(* Logix 5000 project; controller P6 vendor 1 type 14 code 92 rev 20.55; software revision 20.01 *)

TASK MainTask (continuous, watchdog 500 ms) : MainProgram

MODULES
   Local : vendor 1 type 14 code 92 (ICP 0, rev 20.55)
      P6_EN2T_PCN : 1756-EN2T (ICP 1, Ethernet 192.168.1.60, rev 10.1)
         P2 : 1756-EN2T (Ethernet 192.168.1.20, rev 10.1, Output RPI 10 ms)
            P2_CONTROLLER : vendor 1 type 14 code 92 (ICP 0, rev 20.1)
         P1 : 1756-EN2T (Ethernet 192.168.1.10, rev 10.1, Output RPI 10 ms)
            P1_CONTROLLER : vendor 1 type 14 code 92 (ICP 0, rev 20.1)
      P6_EN2TR_RIO : vendor 1 type 12 code 200 (ICP 2, Ethernet 192.168.0.60, rev 10.1)
         RIO6 : 1794-AENTR (Ethernet 192.168.0.62, rev 1.1, Output RPI 20 ms)
            RIO6_DI : 1794-IB32 (Flex 0, rev 1.1, Input RPI 20 ms)
            RIO6_DO : vendor 1 type 7 code 35 (Flex 1, rev 1.1)
            RIO6_AI : 1794-IE12 (Flex 2, rev 1.1, Output RPI 78 ms)
         WRIO6 : vendor 309 type 12 code 1000 (Ethernet 192.168.0.65, rev 3.1, Output RPI 20 ms)
            WRIO6_AI : 1734-IE2C (PointIO 1, rev 3.1, Input RPI 80 ms)
END_MODULES

TYPE AIN_UDT :
STRUCT
   Pv : REAL;
   Heu : REAL;
   Leu : REAL;
   SAHH : REAL;
   SAH : REAL;
   SAL : REAL;
   SALL : REAL;
   AHH : BOOL;
   AH : BOOL;
   AL : BOOL;
   ALL : BOOL;
   Wifi_Enb : BOOL;
   Hty : BOOL;
   Sim : BOOL;
   Sim_PV : REAL;
END_STRUCT
END_TYPE

TYPE AUTOINP_UDT :
STRUCT
   ON : BOOL;
END_STRUCT
END_TYPE

TYPE ControllerLEDStatus :
STRUCT
   Off : BOOL;
   SolidGreen : BOOL;
   FlashingGreen : BOOL;
   SolidYellow : BOOL;
   FlashingYellow : BOOL;
   FlashingRed : BOOL;
   SolidRed : BOOL;
END_STRUCT
END_TYPE

TYPE DOSING_SETPOINT_UDT :
STRUCT
   High_Setpoint : REAL;
   Low_Setpoint : REAL;
END_STRUCT
END_TYPE

TYPE Duty2_UDT :
STRUCT
   Selection : INT;
   Pump_Running : BOOL;
   Selected_Pmp_Not_Avl : BOOL;
   Both_Pmp_Not_Avl : BOOL;
END_STRUCT
END_TYPE

TYPE FaultRecord :
STRUCT
   timelow : DINT;
   timehigh : DINT;
   type : INT;
   code : INT;
   info : DINT[8];
END_STRUCT
END_TYPE

TYPE FIT_UDT :
STRUCT
   Pv : REAL;
   Heu : REAL;
   Leu : REAL;
   SAHH : REAL;
   SAH : REAL;
   SAL : REAL;
   SALL : REAL;
   Totaliser : REAL;
   AHH : BOOL;
   AH : BOOL;
   AL : BOOL;
   ALL : BOOL;
   Sim : BOOL;
   Sim_PV : REAL;
   Wifi_Enb : BOOL;
   Rst_Totaliser : BOOL;
   Hty : BOOL;
END_STRUCT
END_TYPE

TYPE Logix_Status_FP :
STRUCT
   ClearMinorFaults : DINT;
   Sts_MinorFaultEvents : DINT;
   Sts_MinorFaultBits : DINT;
   Sts_Redundant : DINT;
   Set_FaceplateAnimation : DINT;
   Val_ProductCode : DINT;
   MemoryTemp : INT[29];
   Val_raw_data : INT;
   Sts_IO_LED_raw : INT;
   Sts_ProductCode : INT;
   Val_Force_data_raw : INT;
   MemoryRequestData : SINT[12];
   Sts_Force_Installed : BOOL;
   Sts_Force_Enabled : BOOL;
   Sts_Faulted : BOOL;
   Sts_Run : BOOL;
   Sts_Program : BOOL;
   Sts_Minor_fault : BOOL;
   Sts_Major_fault : BOOL;
   Sts_KS_in_run : BOOL;
   Sts_KS_in_program : BOOL;
   Sts_KS_in_remote : BOOL;
   Sts_Changingmodes : BOOL;
   Sts_Test : BOOL;
   Sts_Ladder_Working : BOOL;
   Cmd_ClearFaultRecord : BOOL;
   Set_Controller_Description : STRING;
   UpdateDelayTimer : TIMER;
   Val_MajorFault : FaultRecord;
   Val_MFS : FaultRecord;
   Sts_IO_LED : ControllerLEDStatus;
   Sts_Battery_LED : ControllerLEDStatus;
   MemoryData : Memory_Data;
   TEST : DINT;
END_STRUCT
END_TYPE

TYPE Memory_Data :
STRUCT
   Free_Mem_IO : DINT;
   Free_Mem_DT : DINT;
   Free_Memory : DINT;
   Total_Mem_IO : DINT;
   Total_Mem_DT : DINT;
   Total_Memory : DINT;
   Biggest_IO_Mem_Size_Ava : DINT;
   Biggest_DT_Mem_Size_Ava : DINT;
END_STRUCT
END_TYPE

TYPE MV_UDT :
STRUCT
   Cmd : INT;
   Status : INT;
   Reset : BOOL;
   Auto : BOOL;
   FTO : BOOL;
   FTC : BOOL;
END_STRUCT
END_TYPE

TYPE PLANT_AUTO_UDT :
STRUCT
   ON : BOOL;
   OFF : BOOL;
END_STRUCT
END_TYPE

TYPE PLANT_UDT :
STRUCT
   START : BOOL;
   STOP : BOOL;
END_STRUCT
END_TYPE

TYPE PMP_UDT :
STRUCT
   Cmd : INT;
   Status : INT;
   RunMin : REAL;
   Total_RunMin : REAL;
   RunHr : REAL;
   Total_RunHr : REAL;
   Remote : BOOL;
   Auto : BOOL;
   Fault : BOOL;
   Avl : BOOL;
   Permissive : DINT;
   Shutdown : DINT;
   SD : DINT;
   Reset : BOOL;
   Reset_RunHr : BOOL;
   FTR : BOOL;
   FTS : BOOL;
END_STRUCT
END_TYPE

TYPE PRECONDITION_UDT :
STRUCT
   PERMISSIVE1 : BOOL;
   PERMISSIVE2 : BOOL;
   PERMISSIVE3 : BOOL;
   PERMISSIVE4 : BOOL;
   PERMISSIVE5 : BOOL;
   SHUTDOWN1 : BOOL;
   SHUTDOWN2 : BOOL;
   SHUTDOWN3 : BOOL;
   SHUTDOWN4 : BOOL;
   SHUTDOWN5 : BOOL;
END_STRUCT
END_TYPE

TYPE RED_STAT :
STRUCT
   Redundancy_status_of_the_controller : INT;
   Redundancy_state_of_the_partner : INT;
END_STRUCT
END_TYPE

TYPE SWITCH_UDT :
STRUCT
   Alarm : BOOL;
   Delay : DINT;
END_STRUCT
END_TYPE

TYPE UV_UDT :
STRUCT
   Cmd : INT;
   Status : INT;
   RunMin : REAL;
   Total_RunMin : REAL;
   RunHr : REAL;
   Total_RunHr : REAL;
   Remote : BOOL;
   Auto : BOOL;
   Fault : BOOL;
   Avl : BOOL;
   Permissive : INT;
   Shutdown : INT;
   Reset : BOOL;
   Reset_RunHr : BOOL;
   FT_Start : BOOL;
   FT_Stop : BOOL;
END_STRUCT
END_TYPE

TYPE WIFI_UDT :
STRUCT
   PLC_WIFI : BOOL;
   RIO_WIFI : BOOL;
END_STRUCT
END_TYPE

ADD_ON_INSTRUCTION AIN_FBD   (* revision 1.0 *)
VAR_INPUT
   WRIO_Enb : BOOL; {visible}
   Raw_RIO : INT; {visible}
   Raw_WRIO : INT; {visible}
   L_Raw_RIO : INT; {visible}
   H_Raw_RIO : INT; {visible}
   L_Raw_WRIO : INT; {visible}
   H_Raw_WRIO : INT; {visible}
   HEU : INT; {visible}
   LEU : INT; {visible}
END_VAR
VAR_OUTPUT
   Hty : BOOL; {visible}
   Wifi_Enb : BOOL; {access Read Only, visible}
   AHH : BOOL; {visible}
   AH : BOOL; {access Read Only, visible}
   AL : BOOL; {access Read Only, visible}
   ALL : BOOL; {visible}
END_VAR
VAR_INPUT
   SAHH : REAL; {visible}
   SAH : REAL; {visible}
   SAL : REAL; {visible}
   SALL : REAL; {visible}
   Simulation : BOOL; {visible}
   RIO_Hty : BOOL; {visible}
   WRIO_Hty : BOOL; {visible}
END_VAR
VAR_IN_OUT
   Pv : REAL; {required}
   Sim_PV : REAL; {required}
   HMI : AIN_UDT; {required}
END_VAR
VAR
   SCALE : SCALE; {access None}
   ALM : ALARM; {access None}
   _Raw : INT; {access None}
   _L_Raw : INT; {access None}
   _H_Raw : INT; {access None}
   _Inst_Hty : BOOL; {access None}
END_VAR

ROUTINE Logic   (* structured text *)
   (*RIO and Wireless RIO Selection*)
   
   IF WRIO_Enb THEN
   	Wifi_Enb	:= 1;
   	_Raw		:= Raw_WRIO;
   	_H_Raw		:= H_Raw_WRIO;
   	_L_Raw		:= L_Raw_WRIO;
   	_Inst_Hty 	:= WRIO_Hty;
   ELSE
   	Wifi_Enb	:= 0;
   	_Raw		:= Raw_RIO;
   	_H_Raw		:= H_Raw_RIO;
   	_L_Raw		:= L_Raw_RIO;
   	_Inst_Hty 	:= RIO_Hty;
   END_IF;
   
   (*Calculation for PV*)
   IF Simulation THEN
   	Pv	:=Sim_PV;
   ELSE
   	SCALE.In		:=_Raw;
   	SCALE.InRawMax	:=_H_Raw;
   	SCALE.InRawMin	:=_L_Raw;
   	SCALE.InEUMax	:=HEU;
   	SCALE.InEUMin	:=LEU;
   	SCL(SCALE);
   
   	IF SCALE.Out<0 THEN
   		Pv	:= 0.0;
   	ELSE
   		Pv	:=SCALE.Out;
   	END_IF;
   
   	Sim_PV	:=Pv;
   
   END_IF;
   
   (*Alarms*)
   ALM.In			:=Pv;
   ALM.HHLimit		:=SAHH;
   ALM.HLimit		:=SAH;
   ALM.LLimit		:=SAL;
   ALM.LLLimit		:=SALL;
   ALM(ALM);
   
   AHH				:=ALM.HHAlarm;
   AH				:=ALM.HAlarm;
   AL				:=ALM.LAlarm;
   ALL				:=ALM.LLAlarm;
   
   Hty:= _Inst_Hty AND (_Raw > _L_Raw) AND (_Raw < _H_Raw)  ;
   
   
   
   
   
   
END_ROUTINE
END_ADD_ON_INSTRUCTION

ADD_ON_INSTRUCTION Duty2_FBD   (* revision 1.0 *)
VAR_INPUT
   AutoInp : BOOL; {visible}
   Selection : INT; {visible}
END_VAR
VAR_OUTPUT
   Start_Pmp1 : BOOL; {visible}
   Start_Pmp2 : BOOL; {visible}
END_VAR
VAR_IN_OUT
   PMP1 : PMP_UDT; {required}
   PMP2 : PMP_UDT; {required}
   HMI : Duty2_UDT; {required}
END_VAR

ROUTINE Logic   (* structured text *)
   IF PMP1.Status=2 OR PMP2.Status=2 THEN
   	HMI.Pump_Running := 1;
   ELSE
   	HMI.Pump_Running := 0;
   END_IF;
   
   HMI.Both_Pmp_Not_Avl		:= NOT PMP1.Avl AND NOT PMP2.Avl;
   
   IF AutoInp THEN
   	CASE Selection OF
   		(*PUMP 1 *)
   		1:
   			IF PMP1.Avl THEN
   				Start_Pmp1					:=1;
   				Start_Pmp2					:=0;
   				HMI.Selected_Pmp_Not_Avl	:=0;
   			ELSIF NOT PMP1.Avl AND PMP2.Avl THEN
   				Start_Pmp1					:=0;
   				Start_Pmp2					:=1;
   				HMI.Selected_Pmp_Not_Avl	:=1;
   			ELSIF NOT PMP1.Avl AND NOT PMP2.Avl	THEN
   				Start_Pmp1					:=0;
   				Start_Pmp2					:=0;
   			ELSE
   				HMI.Selected_Pmp_Not_Avl	:=0;
   			END_IF;
   
   		(*PUMP 2 *)
   		2:
   			IF PMP2.Avl THEN
   				Start_Pmp1					:=0;
   				Start_Pmp2					:=1;
   				HMI.Selected_Pmp_Not_Avl	:=0;
   			ELSIF NOT PMP2.Avl AND PMP1.Avl THEN
   				Start_Pmp1					:=1;
   				Start_Pmp2					:=0;
   				HMI.Selected_Pmp_Not_Avl	:=1;
   			ELSIF NOT PMP1.Avl AND NOT PMP2.Avl	THEN
   				Start_Pmp1					:=0;
   				Start_Pmp2					:=0;
   			ELSE
   				HMI.Selected_Pmp_Not_Avl	:=0;
   			END_IF;
   	END_CASE;
   ELSE
   	Start_Pmp1					:=0;
   	Start_Pmp2					:=0;
   END_IF;
   
   
END_ROUTINE
END_ADD_ON_INSTRUCTION

ADD_ON_INSTRUCTION FIT_FBD   (* revision 1.0 *)
VAR_INPUT
   WRIO_Enb : BOOL; {visible}
   Raw_RIO : INT; {visible}
   Raw_WRIO : INT; {visible}
   L_Raw_RIO : INT; {visible}
   H_Raw_RIO : INT; {visible}
   L_Raw_WRIO : INT; {visible}
   H_Raw_WRIO : INT; {visible}
   HEU : REAL; {visible}
   LEU : REAL; {visible}
END_VAR
VAR_OUTPUT
   Hty : BOOL; {visible}
   Wifi_Enb : BOOL; {visible}
   AHH : BOOL; {visible}
   AH : BOOL; {access Read Only, visible}
   AL : BOOL; {access Read Only, visible}
   ALL : BOOL; {visible}
END_VAR
VAR_INPUT
   SAHH : REAL; {visible}
   SAH : REAL; {visible}
   SAL : REAL; {visible}
   SALL : REAL; {visible}
   Simulation : BOOL; {visible}
   RIO_Hty : BOOL; {visible}
   WRIO_Hty : BOOL; {visible}
   Totaliser_Enb : BOOL; {visible}
   Rst_Totaliser : BOOL; {visible}
END_VAR
VAR_IN_OUT
   Totaliser : REAL; {required}
   Pv : REAL; {required}
   Sim_Pv : REAL; {required}
   HMI : FIT_UDT; {required}
END_VAR
VAR
   SCALE : SCALE; {access None}
   ALM : ALARM; {access None}
   TON : FBD_TIMER; {access None}
   _SEC_P : BOOL; {access None}
   _Inst_Hty : BOOL; {access None}
   _L_Raw : INT; {access None}
   _H_Raw : INT; {access None}
   _Raw : INT; {access None}
   R_TRIG : FBD_ONESHOT; {access None}
END_VAR

ROUTINE Logic   (* structured text *)
   (*RIO and Wireless RIO Selection*)
   
   IF WRIO_Enb THEN
   	Wifi_Enb	:= 1;
   	_Raw		:= Raw_WRIO;
   	_H_Raw		:= H_Raw_WRIO;
   	_L_Raw		:= L_Raw_WRIO;
   	_Inst_Hty 	:= WRIO_Hty;
   ELSE
   	Wifi_Enb	:= 0;
   	_Raw		:= Raw_RIO;
   	_H_Raw		:= H_Raw_RIO;
   	_L_Raw		:= L_Raw_RIO;
   	_Inst_Hty 	:= RIO_Hty;
   END_IF;
   
   (*Calculation for PV*)
   IF Simulation THEN
   	Pv	:= Sim_Pv   ;
   ELSE
   	SCALE.In		:=_Raw;
   	SCALE.InRawMax	:=_H_Raw;
   	SCALE.InRawMin	:=_L_Raw;
   	SCALE.InEUMax	:=HEU;
   	SCALE.InEUMin	:=LEU;
   	SCL(SCALE);
   	IF SCALE.Out>0 THEN
   		Pv	:=SCALE.Out;
   	ELSIF SCALE.Out<=0 THEN
   		Pv	:=0.0;
   	END_IF;
   
   	Sim_Pv	:=Pv;
   END_IF;
   
   (*Alarms*)
   ALM.In			:=Pv;
   ALM.HHLimit		:=SAHH;
   ALM.HLimit		:=SAH;
   ALM.LLimit		:=SAL;
   ALM.LLLimit		:=SALL;
   ALM(ALM);
   
   AHH				:=ALM.HHAlarm;
   AH				:=ALM.HAlarm;
   AL				:=ALM.LAlarm;
   ALL				:=ALM.LLAlarm;
   
   (*SECOND PULSE*)
   TON.PRE	:=1000;
   TON.TimerEnable	:=1;
   TONR(TON );
   R_TRIG.InputBit :=TON.DN ;
   OSRI( R_TRIG);
   _SEC_P  := R_TRIG.OutputBit;
   TON.Reset := _SEC_P;
   
   IF Totaliser_Enb THEN
   	IF _SEC_P THEN
   		HMI.Totaliser := HMI.Totaliser +  (ABS(Pv) / 3600 );
   	END_IF;
   END_IF;
   
   IF  Rst_Totaliser   THEN
   	HMI.Totaliser	:=0;
   END_IF;
   
   Hty:= _Inst_Hty AND (_Raw > _L_Raw) AND (_Raw < _H_Raw)  ;
   
   
   
   
   
   
END_ROUTINE
END_ADD_ON_INSTRUCTION

ADD_ON_INSTRUCTION MV_FBD   (* revision 1.0 *)
VAR_INPUT
   Auto : BOOL; {visible}
END_VAR
VAR_OUTPUT
   Cmd_Open : BOOL; {visible}
   Cmd_Close : BOOL; {visible}
   FTO : BOOL; {visible}
   FTC : BOOL; {access Read Only, visible}
END_VAR
VAR_INPUT
   AutoInp : BOOL; {visible}
   ZSO : BOOL; {visible}
   Open_TM : DINT; {visible}
   ZSC : BOOL; {visible}
   Close_TM : DINT; {visible}
END_VAR
VAR_IN_OUT
   Cmd : INT; {required}
   HMI : MV_UDT; {required}
END_VAR
VAR
   TON_Open_TM : FBD_TIMER; {access None}
   TON_Close_TM : FBD_TIMER; {access None}
END_VAR

ROUTINE Logic   (* structured text *)
   (*Fail to Close*)
   TON_Close_TM.PRE 			:= 	Close_TM*1000;
   TON_Close_TM.TimerEnable 	:=  Cmd_Close;
   TONR(TON_Close_TM);
   
   (*Fail to Open*)
   TON_Open_TM.PRE 			:= 	Open_TM*1000;
   TON_Open_TM.TimerEnable 	:= 	Cmd_Open;
   TONR(TON_Open_TM);
   
   IF ZSC THEN
   	HMI.Status	:=1;
   ELSIF ZSO THEN
   	HMI.Status	:=2;
   ELSE
   	HMI.Status	:=0;
   END_IF;
   
   
   IF HMI.Reset THEN
   	(*IF NOT TON_Close_TM.DN AND ZSC THEN*)
   			FTC		:= 0;
   	(*END_IF;*)
   	(*IF NOT TON_Open_TM.DN AND ZSO THEN*)
   			FTO		:= 0;
   	(*END_IF;*)
   END_IF;
   
   IF  NOT Auto THEN
   	CASE HMI.Cmd OF
   		1:	(*CLOSE*)
   			Cmd_Close	:= 1;
   			Cmd_Open	:= 0;
   			IF TON_Close_TM.DN AND (NOT ZSC) THEN
   				FTC		:= 1;
   				FTO		:= 0;
   			END_IF;
   		2:	(*OPEN*)
   			IF FTO OR FTC    THEN
   				HMI.Cmd := 1;
   			END_IF;
   
   			IF NOT FTC AND NOT FTO THEN
   				Cmd_Close	:= 0;
   				Cmd_Open	:= 1;
   			END_IF;
   
   			IF TON_Open_TM.DN AND (NOT ZSO) THEN
   				FTC		:= 0;
   				FTO		:= 1;
   				HMI.Cmd := 1;
   			END_IF;
   	END_CASE;
   ELSE
   	(*Maintain Last status when switching from Auto to Manual*)
   	IF ZSO THEN
   		Cmd	:= 2;
   	END_IF;
   	IF ZSC THEN
   		Cmd	:= 1;
   	END_IF;
   
   	IF  AutoInp  THEN
   		Cmd_Close	:= 0;
   		Cmd_Open	:= 1;
   		IF TON_Open_TM.DN AND (NOT ZSO) THEN
   			FTC		:= 0;
   			FTO		:= 1;
   		END_IF;
   	ELSE
   		Cmd_Close	:= 1;
   		Cmd_Open	:= 0;
   		IF TON_Close_TM.DN AND (NOT ZSC) THEN
   			FTC		:= 1;
   			FTO		:= 0;
   		END_IF;
   	END_IF;
   END_IF;
   
   
END_ROUTINE
END_ADD_ON_INSTRUCTION

ADD_ON_INSTRUCTION PMP_FBD   (* revision 1.0 *)
VAR_OUTPUT
   Cmd_Start : BOOL; {visible}
   Avl : BOOL; {visible}
   Fault : BOOL; {visible}
   FT_Stop : BOOL; {visible}
   FT_Start : BOOL; {visible}
   RunHr : REAL; {visible}
   Total_RunHr : REAL; {visible}
   SD : DINT; {access Read Only, visible}
END_VAR
VAR_INPUT
   Auto : BOOL; {visible}
   AutoInp : BOOL; {visible}
   Remote : BOOL; {visible}
   Run : BOOL; {visible}
   Trip : BOOL; {visible}
   Start_TM : DINT; {visible}
   Stop_TM : DINT; {visible}
   Rst : BOOL; {visible}
   Rst_RunHr : BOOL; {visible}
   Permissive : DINT; {visible}
   Shutdown : DINT; {visible}
END_VAR
VAR_IN_OUT
   RunMin : REAL; {required}
   Total_RunMin : REAL; {required}
   Cmd : INT; {required}
   HMI : PMP_UDT; {required}
END_VAR
VAR
   TON_Start_TM : FBD_TIMER; {access None}
   TON_Stop_TM : FBD_TIMER; {access None}
   _Min_P : BOOL; {access None}
   TON_Min : FBD_TIMER; {access None}
   R_TRIG_SEC : FBD_ONESHOT; {access None}
END_VAR

ROUTINE Logic   (* structured text *)
   (*Fail to Start*)
   TON_Start_TM.PRE 			:= 	Start_TM*1000;
   TON_Start_TM.TimerEnable 	:=  Cmd_Start;
   TONR(TON_Start_TM);
   
   (*Fail to Stop*)
   TON_Stop_TM.PRE 			:= 	Stop_TM*1000;
   TON_Stop_TM.TimerEnable 	:=  NOT Cmd_Start;
   TONR(TON_Stop_TM);
   
   IF (NOT Run) THEN
   	HMI.Status	:=1;
   ELSE
   	HMI.Status	:=2;
   END_IF;
   
   IF Fault THEN
   	HMI.Fault:= 1;
   ELSE
   	HMI.Fault:= 0;
   END_IF;
   
   IF HMI.Reset THEN
   	IF NOT TON_Stop_TM.DN THEN
   			FT_Stop		:= 0;
   	END_IF;
   	IF NOT TON_Start_TM.DN THEN
   			FT_Start	:= 0;
   	END_IF;
   
   	SD :=0;
   
   END_IF;
   
   Fault		:=Trip OR SD<>0;
   HMI.Remote	:=Remote;
   Avl:= Auto AND Remote AND NOT Fault AND NOT FT_Start AND NOT FT_Stop AND SD=0 ;
   
   IF Remote THEN
   	IF  NOT Auto THEN
   		CASE HMI.Cmd OF
   			1:	(*Stop*)
   				Cmd_Start	:=0;
   				IF TON_Stop_TM.DN AND Run THEN
   					FT_Start	:= 0;
   					FT_Stop		:= 1;
   				END_IF;
   			2:	(*OPEN*)
   				IF NOT Fault AND NOT FT_Start AND NOT FT_Stop AND (Permissive=-1) AND HMI.SD=0 THEN
   					Cmd_Start	:= 1;
   				ELSIF Cmd_Start AND (HMI.SD<>0) OR Fault THEN
   					SD				:= HMI.SD;
   					Cmd_Start		:= 0;
   					HMI.Cmd 		:= 1;
   				ELSIF (Permissive<>-1) THEN
   					HMI.Cmd 		:= 1;
   				END_IF;
   
   				IF TON_Start_TM.DN AND NOT Run THEN
   					FT_Start	:= 1;
   					FT_Stop		:= 0;
   					Cmd_Start	:= 0;
   					HMI.Cmd 	:= 1;
   				END_IF;
   		END_CASE;
   	ELSE
   		IF Run THEN
   			Cmd	:= 2;
   		END_IF;
   		IF (NOT Run) OR Fault OR FT_Start OR FT_Stop THEN
   			Cmd	:= 1;
   		END_IF;
   
   		IF  AutoInp  THEN
   			IF NOT Fault AND NOT FT_Start AND NOT FT_Stop AND (Permissive=-1) AND HMI.SD=0  THEN
   				Cmd_Start	:=1;
   			ELSIF Cmd_Start OR (HMI.SD<>0) OR Fault THEN
   				SD			:= HMI.SD;
   				Cmd_Start	:=0;
   			END_IF;
   
   			IF TON_Start_TM.DN AND NOT Run THEN
   				FT_Start	:= 1;
   				FT_Stop		:= 0;
   				Cmd_Start	:= 0;
   				HMI.Cmd 	:= 1;
   			END_IF;
   		ELSE
   			Cmd_Start	:=0;
   			IF TON_Stop_TM.DN AND Run THEN
   				FT_Start	:= 0;
   				FT_Stop		:= 1;
   
   			END_IF;
   		END_IF;
   	END_IF;
   
   ELSE (*Local*)
   	Cmd_Start	:=0;
   	Cmd	:= 1;
   
   	FT_Start	:= 0;
   	FT_Stop		:= 0;
   
   
   
   
   	(*	IF Run THEN
   			Cmd	:= 2;
   		END_IF;
   		IF (NOT Run) OR Fault OR FT_Start OR FT_Stop THEN
   			Cmd	:= 1;
   		END_IF;
   		*)
   END_IF;
   
   (*1 MIN PULSE*)
   TON_Min.PRE	:=60000;
   TON_Min.TimerEnable	:=1;
   TONR(TON_Min );
   R_TRIG_SEC.InputBit :=TON_Min.DN ;
   OSRI( R_TRIG_SEC);
   _Min_P  := R_TRIG_SEC.OutputBit;
   TON_Min.Reset 	:= _Min_P;
   
   IF Run THEN
   	IF _Min_P THEN
   		RunMin 			:=RunMin + 1.0;
   		Total_RunMin	:=Total_RunMin + 1.0;
   	END_IF;
   END_IF;
   
   RunHr 				:=RunMin/60.0;
   Total_RunHr			:=Total_RunMin/60.0;
   
   IF  Rst_RunHr THEN
   	RunMin	:=0;
   END_IF;
   
   
   
END_ROUTINE
END_ADD_ON_INSTRUCTION

ADD_ON_INSTRUCTION SWITCH_FBD   (* revision 1.0 *)
VAR_INPUT
   Alarm : BOOL; {visible}
   Delay : DINT; {required}
END_VAR
VAR_OUTPUT
   Status : BOOL; {access None, required}
END_VAR
VAR_IN_OUT
   HMI : SWITCH_UDT; {required}
END_VAR
VAR
   TON_Delay_Sec : FBD_TIMER; {access None}
END_VAR

ROUTINE Logic   (* structured text *)
   (*Delay for Alarm*)
   TON_Delay_Sec.PRE 			:= 	Delay*1000;
   TON_Delay_Sec.TimerEnable 	:=  Alarm;
   TONR(TON_Delay_Sec);
   
   Status := TON_Delay_Sec.DN ;
END_ROUTINE
END_ADD_ON_INSTRUCTION

ADD_ON_INSTRUCTION UV_FBD   (* revision 1.0 *)
VAR_OUTPUT
   Cmd_Start : BOOL; {visible}
   Avl : BOOL; {visible}
   Fault : BOOL; {visible}
   FT_Stop : BOOL; {visible}
   FT_Start : BOOL; {visible}
   RunHr : REAL; {visible}
   Total_RunHr : REAL; {visible}
END_VAR
VAR_INPUT
   Auto : BOOL; {visible}
   AutoInp : BOOL; {visible}
   Remote : BOOL; {visible}
   Run : BOOL; {visible}
   Trip : BOOL; {visible}
   Start_TM : DINT; {visible}
   Stop_TM : DINT; {visible}
   Rst : BOOL; {visible}
   Rst_RunHr : BOOL; {visible}
   Permissive : INT; {visible}
   Shutdown : INT; {visible}
END_VAR
VAR_IN_OUT
   RunMin : REAL; {required}
   Total_RunMin : REAL; {required}
   Cmd : INT; {required}
   HMI : UV_UDT; {required}
END_VAR
VAR
   TON_Start_TM : FBD_TIMER; {access None}
   TON_Stop_TM : FBD_TIMER; {access None}
   _Min_P : BOOL; {access None}
   TON_Min : FBD_TIMER; {access None}
   R_TRIG_SEC : FBD_ONESHOT; {access None}
END_VAR

ROUTINE Logic   (* structured text *)
   (*Fail to Start*)
   TON_Start_TM.PRE 			:= 	Start_TM*1000;
   TON_Start_TM.TimerEnable 	:=  Cmd_Start;
   TONR(TON_Start_TM);
   
   (*Fail to Stop*)
   TON_Stop_TM.PRE 			:= 	Stop_TM*1000;
   TON_Stop_TM.TimerEnable 	:=  NOT Cmd_Start;
   TONR(TON_Stop_TM);
   
   IF (NOT Run) THEN
   	HMI.Status	:=1;
   ELSE
   	HMI.Status	:=2;
   END_IF;
   
   IF Fault THEN
   	HMI.Fault:= 1;
   ELSE
   	HMI.Fault:= 0;
   END_IF;
   
   IF HMI.Reset THEN
   	IF NOT TON_Stop_TM.DN THEN
   			FT_Stop		:= 0;
   	END_IF;
   	IF NOT TON_Start_TM.DN THEN
   			FT_Start	:= 0;
   	END_IF;
   END_IF;
   
   
   HMI.Remote	:=Remote;
   Avl:= Auto AND Remote AND NOT Fault AND NOT FT_Stop AND NOT FT_Stop   ;
   
   
   
   IF Remote THEN
   	IF  NOT Auto THEN
   		CASE HMI.Cmd OF
   			1:	(*Stop*)
   				Cmd_Start	:=0;
   				IF TON_Stop_TM.DN AND Run THEN
   					FT_Start	:= 0;
   					FT_Stop		:= 1;
   				END_IF;
   			2:	(*OPEN*)
   				IF NOT Fault AND (NOT FT_Start OR FT_Stop) AND (Permissive=-1) THEN
   					Cmd_Start	:= 1;
   				END_IF;
   
   				IF (Shutdown<>0) OR Fault THEN
   					Cmd_Start	:= 0;
   					HMI.Cmd 	:= 1;
   				END_IF;
   
   				IF TON_Start_TM.DN AND NOT Run THEN
   					FT_Start	:= 1;
   					FT_Stop		:= 0;
   					Cmd_Start	:= 0;
   					HMI.Cmd 	:= 1;
   				END_IF;
   		END_CASE;
   	ELSE
   		IF Run THEN
   			Cmd	:= 2;
   		END_IF;
   		IF (NOT Run) OR Fault OR FT_Start OR FT_Stop THEN
   			Cmd	:= 1;
   		END_IF;
   
   		IF  AutoInp  THEN
   			IF NOT Fault AND (NOT FT_Start OR FT_Stop) AND (Permissive=-1) THEN
   				Cmd_Start	:=1;
   			END_IF;
   
   			IF (Shutdown<>0) OR Fault THEN
   				Cmd_Start	:=0;
   			END_IF;
   
   			IF TON_Start_TM.DN AND NOT Run THEN
   				FT_Start	:= 1;
   				FT_Stop		:= 0;
   				Cmd_Start	:= 0;
   				HMI.Cmd 	:= 1;
   			END_IF;
   		ELSE
   			Cmd_Start	:=0;
   			IF TON_Stop_TM.DN AND Run THEN
   				FT_Start	:= 0;
   				FT_Stop		:= 1;
   
   			END_IF;
   		END_IF;
   	END_IF;
   
   ELSE (*Local*)
   	Cmd_Start	:=0;
   	Cmd	:= 1;
   
   	(*	IF Run THEN
   			Cmd	:= 2;
   		END_IF;
   		IF (NOT Run) OR Fault OR FT_Start OR FT_Stop THEN
   			Cmd	:= 1;
   		END_IF;
   		*)
   END_IF;
   
   (*1 MIN PULSE*)
   TON_Min.PRE	:=60000;
   TON_Min.TimerEnable	:=1;
   TONR(TON_Min );
   R_TRIG_SEC.InputBit :=TON_Min.DN ;
   OSRI( R_TRIG_SEC);
   _Min_P  := R_TRIG_SEC.OutputBit;
   TON_Min.Reset 	:= _Min_P;
   
   IF Run THEN
   	IF _Min_P THEN
   		RunMin 			:=RunMin + 1.0;
   		Total_RunMin	:=Total_RunMin + 1.0;
   	END_IF;
   END_IF;
   
   RunHr 				:=RunMin/60.0;
   Total_RunHr			:=Total_RunMin/60.0;
   
   IF  Rst_RunHr THEN
   	RunMin	:=0;
   END_IF;
   
   
   
END_ROUTINE
END_ADD_ON_INSTRUCTION

VAR_GLOBAL   (* controller tags *)
   _FIT601_Tot_Enb : BOOL;
   _MV301_AutoInp : BOOL;
   _MV302_AutoInp : BOOL;
   _MV303_AutoInp : BOOL;
   _MV304_AutoInp : BOOL;
   _P301_AutoInp : BOOL;
   _P302_AutoInp : BOOL;
   _P401_AutoInp : BOOL;
   _P402_AutoInp : BOOL;
   _P403_AutoInp : BOOL;
   _P404_AutoInp : BOOL;
   _P601_AutoInp : BOOL;
   _P602_AutoInp : BOOL;
   _P603_AutoInp : BOOL;
   _P_BACKWASH_SR : DOMINANT_SET;
   _P_CIP_SR : DOMINANT_SET;
   _P_NAHSO3_ORP_DUTY_AutoInp : BOOL;
   _P_NAHSO3_ORP_DUTY_SR : DOMINANT_SET := (Reset := 1, OutNot := 1);
   _P_PERMEATE_SR : DOMINANT_SET := (OutNot := 1);
   _P_RO_FEED_DUTY_AutoInp : BOOL;
   _P_RO_FEED_DUTY_SR : DOMINANT_SET := (Set := 1, Out := 1);
   _P_UF_FEED_DUTY_AutoInp : BOOL := 1;
   _UV401_AutoInp : BOOL := 1;
   _UV_SR : DOMINANT_SET := (Set := 1, Out := 1);
   AI_AIT_401_HRDNSS : INT := -11;
   AI_AIT_401_HRDNSS_HTY : BOOL := 1;
   AI_AIT_402_ORP : INT := -17;
   AI_AIT_402_ORP_HTY : BOOL := 1;
   AI_DPIT_301_DPRESS : INT;
   AI_DPIT_301_DPRESS_HTY : BOOL;
   AI_FIT_301_FLOW : INT;
   AI_FIT_301_FLOW_HTY : BOOL;
   AI_FIT_401_FLOW : INT := -19;
   AI_FIT_401_FLOW_HTY : BOOL := 1;
   AI_FIT_601_FLOW : INT := -3;
   AI_FIT_601_FLOW_HTY : BOOL := 1;
   AI_LIT_301_LEVEL : INT;
   AI_LIT_301_LEVEL_HTY : BOOL;
   AI_LIT_401_LEVEL : INT := -9;
   AI_LIT_401_LEVEL_HTY : BOOL := 1;
   AI_RIO6_SPARE_01 : INT := -7702;
   AI_RIO6_SPARE_01_HTY : BOOL := 1;
   AI_RIO6_SPARE_02 : INT := -7703;
   AI_RIO6_SPARE_02_HTY : BOOL := 1;
   AI_RIO6_SPARE_03 : INT := -7702;
   AI_RIO6_SPARE_03_HTY : BOOL := 1;
   AI_RIO6_SPARE_04 : INT := -7703;
   AI_RIO6_SPARE_04_HTY : BOOL := 1;
   AI_RIO6_SPARE_05 : INT := -7704;
   AI_RIO6_SPARE_05_HTY : BOOL := 1;
   AI_RIO6_SPARE_06 : INT := -7702;
   AI_RIO6_SPARE_06_HTY : BOOL := 1;
   AI_RIO6_SPARE_07 : INT := -7704;
   AI_RIO6_SPARE_07_HTY : BOOL := 1;
   AI_RIO6_SPARE_08 : INT := -7703;
   AI_RIO6_SPARE_08_HTY : BOOL := 1;
   AI_RIO6_SPARE_09 : INT := -7702;
   AI_RIO6_SPARE_09_HTY : BOOL := 1;
   AI_RIO6_SPARE_10 : INT := -7702;
   AI_RIO6_SPARE_10_HTY : BOOL := 1;
   AI_RIO6_SPARE_11 : INT := -7704;
   AI_RIO6_SPARE_11_HTY : BOOL := 1;
   AIT401_FB : AIN_FBD := (Raw_RIO := -11, Raw_WRIO := 3266, H_Raw_RIO := 31208, L_Raw_WRIO := 3277, H_Raw_WRIO := 16383, HEU := 2, Hty := 1, AL := 1, ALL := 1, RIO_Hty := 1);
   AIT401_FB_01 : AIN_FBD;
   AIT402_FB : AIN_FBD := (Raw_RIO := -17, Raw_WRIO := 3268, H_Raw_RIO := 31208, L_Raw_WRIO := 3277, H_Raw_WRIO := 16383, HEU := 2, Hty := 1, AL := 1, ALL := 1, RIO_Hty := 1);
   DI_DPSH_301_HIGH : BOOL;
   DI_LS_401_LOW : BOOL;
   DI_LS_601_HIGH : BOOL := 1;
   DI_LS_601_LOW : BOOL;
   DI_LS_602_HIGH : BOOL := 1;
   DI_LS_602_LOW : BOOL;
   DI_LS_603_HIGH : BOOL;
   DI_LS_603_LOW : BOOL := 1;
   DI_P_404_RUN : BOOL;
   DI_P_601_AUTO : BOOL := 1;
   DI_P_601_FAULT : BOOL;
   DI_P_601_RUN : BOOL;
   DI_P_602_AUTO : BOOL := 1;
   DI_P_602_FAULT : BOOL;
   DI_P_602_RUN : BOOL;
   DI_P_603_AUTO : BOOL := 1;
   DI_P_603_FAULT : BOOL;
   DI_P_603_RUN : BOOL;
   DI_PSH_301_HIGH : BOOL;
   DI_RIO6_SPARE_10 : BOOL;
   DI_RIO6_SPARE_11 : BOOL;
   DI_RIO6_SPARE_12 : BOOL;
   DI_RIO6_SPARE_13 : BOOL;
   DI_RIO6_SPARE_14 : BOOL;
   DI_RIO6_SPARE_15 : BOOL;
   DI_RIO6_SPARE_16 : BOOL;
   DI_RIO6_SPARE_17 : BOOL;
   DI_RIO6_SPARE_18 : BOOL;
   DI_RIO6_SPARE_19 : BOOL;
   DI_RIO6_SPARE_20 : BOOL;
   DI_RIO6_SPARE_21 : BOOL;
   DI_RIO6_SPARE_22 : BOOL;
   DI_RIO6_SPARE_23 : BOOL;
   DI_RIO6_SPARE_24 : BOOL;
   DI_RIO6_SPARE_25 : BOOL;
   DI_RIO6_SPARE_26 : BOOL;
   DI_RIO6_SPARE_27 : BOOL;
   DI_RIO6_SPARE_28 : BOOL;
   DI_RIO6_SPARE_29 : BOOL;
   DI_RIO6_SPARE_30 : BOOL;
   DI_RIO6_SPARE_31 : BOOL;
   DI_UV_401_AUTO : BOOL := 1;
   DI_UV_401_FAULT : BOOL;
   DI_UV_401_RUN : BOOL;
   DI_WIFI_PLC_6 : BOOL;
   DI_WIFI_RIO_6 : BOOL;
   DO_P_601_START : BOOL;
   DO_P_602_START : BOOL;
   DO_P_603_START : BOOL;
   DO_RIO6_SPARE_04 : BOOL;
   DO_RIO6_SPARE_05 : BOOL;
   DO_RIO6_SPARE_06 : BOOL;
   DO_RIO6_SPARE_07 : BOOL;
   DO_RIO6_SPARE_08 : BOOL;
   DO_RIO6_SPARE_09 : BOOL;
   DO_RIO6_SPARE_10 : BOOL;
   DO_RIO6_SPARE_11 : BOOL;
   DO_RIO6_SPARE_12 : BOOL;
   DO_RIO6_SPARE_13 : BOOL;
   DO_RIO6_SPARE_14 : BOOL;
   DO_RIO6_SPARE_15 : BOOL;
   DPIT301_FB : AIN_FBD := (WRIO_Enb := 1, L_Raw_RIO := 6242, H_Raw_RIO := 31208, L_Raw_WRIO := 3277, H_Raw_WRIO := 16383, HEU := 2, Wifi_Enb := 1, AL := 1, ALL := 1);
   DPSH301_FB : SWITCH_FBD;
   FIT102_FB : FIT_FBD;
   FIT301_FB : FIT_FBD := (WRIO_Enb := 1, L_Raw_RIO := 6242, H_Raw_RIO := 31208, L_Raw_WRIO := 3277, H_Raw_WRIO := 16383, HEU := 2.0, Wifi_Enb := 1, AL := 1, ALL := 1);
   FIT401_FB : FIT_FBD := (Raw_RIO := -19, Raw_WRIO := 3263, L_Raw_RIO := 6242, H_Raw_RIO := 31208, L_Raw_WRIO := 3277, H_Raw_WRIO := 16383, HEU := 5.0, Hty := 1, AL := 1, ALL := 1, RIO_Hty := 1);
   FIT601_FB : FIT_FBD := (Raw_RIO := -3, L_Raw_RIO := -5, H_Raw_RIO := 31208, L_Raw_WRIO := 3277, H_Raw_WRIO := 16383, HEU := 2.0, Hty := 1, AL := 1, ALL := 1, SAHH := 3.0, SAH := 2.0, SAL := 1.0, SALL := 0.5, RIO_Hty := 1, WRIO_Hty := 1);
   HMI_AIT202 : AIN_UDT := (Pv := 7.3255577, SAHH := 12.0, SAH := 7.05, SAL := 6.95, SALL := 3.0, AH := 1, Hty := 1, Sim_PV := 7.3255577);
   HMI_FIT301 : FIT_UDT := (Totaliser := -0.09362481, AL := 1, ALL := 1, Wifi_Enb := 1);
   HMI_FIT401 : FIT_UDT := (Pv := -1.2539053, Totaliser := -0.9073935, AL := 1, ALL := 1, Hty := 1);
   HMI_FIT601 : FIT_UDT := (Pv := 0.00012815173, SAHH := 3.0, SAH := 2.0, SAL := 1.0, SALL := 0.5, Totaliser := 0.8749698, AL := 1, ALL := 1, Sim_PV := 0.00012815173, Hty := 1);
   HMI_LIT101 : AIN_UDT := (Pv := 812.6106, SAHH := 1000.0, SAH := 800.0, SAL := 500.0, SALL := 250.0, AH := 1, Hty := 1, Sim_PV := 812.6106);
   HMI_LIT301 : AIN_UDT := (Pv := -0.5000763, AL := 1, ALL := 1, Wifi_Enb := 1);
   HMI_LIT401 : AIN_UDT := (Pv := -0.0005767752, AL := 1, ALL := 1, Hty := 1);
   HMI_LS401 : SWITCH_UDT;
   HMI_LSH601 : SWITCH_UDT := (Alarm := 1);
   HMI_LSH602 : SWITCH_UDT := (Alarm := 1);
   HMI_LSH603 : SWITCH_UDT;
   HMI_LSL601 : SWITCH_UDT;
   HMI_LSL602 : SWITCH_UDT;
   HMI_LSL603 : SWITCH_UDT := (Alarm := 1);
   HMI_NAHSO3_ORP_DOSING : DOSING_SETPOINT_UDT;
   HMI_P301 : PMP_UDT := (Cmd := 1, Status := 1, Remote := 1, Permissive := -1);
   HMI_P302 : PMP_UDT := (Cmd := 1, Status := 1, Remote := 1, Permissive := -1);
   HMI_P401 : PMP_UDT := (Status := 1, Remote := 1, Permissive := -1);
   HMI_P402 : PMP_UDT := (Status := 1, Remote := 1, Permissive := -1);
   HMI_P403 : PMP_UDT := (Status := 1, Remote := 1, Permissive := -1);
   HMI_P404 : PMP_UDT := (Status := 1, Remote := 1, Permissive := -1);
   HMI_P501 : PMP_UDT;
   HMI_P502 : PMP_UDT;
   HMI_P601 : PMP_UDT := (Cmd := 1, Status := 1, RunMin := 2166.0, Total_RunMin := 2166.0, RunHr := 36.1, Total_RunHr := 36.1, Remote := 1, Auto := 1, Avl := 1, Permissive := -1, Reset := 1);
   HMI_P601_MSG : PRECONDITION_UDT := (PERMISSIVE1 := 1);
   HMI_P602 : PMP_UDT := (Cmd := 1, Status := 1, RunMin := 63.0, Total_RunMin := 63.0, RunHr := 1.05, Total_RunHr := 1.05, Remote := 1, Auto := 1, Avl := 1, Permissive := -1, Reset := 1);
   HMI_P602_MSG : PRECONDITION_UDT := (PERMISSIVE1 := 1);
   HMI_P603 : PMP_UDT := (Cmd := 1, Status := 1, Remote := 1, Auto := 1, Avl := 1, Permissive := -2, SD := 1, Reset := 1);
   HMI_P603_MSG : PRECONDITION_UDT;
   HMI_P6_PERMISSIVE : AUTOINP_UDT := (ON := 1);
   HMI_P6_STATE : INT := 1;
   HMI_P_NAHSO3_ORP_DUTY : Duty2_UDT;
   HMI_P_RO_FEED_DUTY : Duty2_UDT;
   HMI_P_UF_FEED_DUTY : Duty2_UDT;
   HMI_PLANT : PLANT_UDT;
   HMI_PLANT_AUTO : PLANT_AUTO_UDT;
   HMI_PLANT_PERMISSIVE : BOOL := 1;
   HMI_PLANT_RESET : PLANT_AUTO_UDT;
   HMI_PSH301 : SWITCH_UDT;
   HMI_START_PLANT : BOOL;
   HMI_STOP_PLANT : BOOL;
   HMI_UV401 : UV_UDT := (Cmd := 1, Status := 1, Remote := 1, Permissive := -1);
   HMI_WIFI : WIFI_UDT;
   LIT301_FB : AIN_FBD := (WRIO_Enb := 1, L_Raw_RIO := 6242, H_Raw_RIO := 31208, L_Raw_WRIO := 3277, H_Raw_WRIO := 16383, HEU := 2, Wifi_Enb := 1, AL := 1, ALL := 1);
   LIT401_FB : AIN_FBD := (Raw_RIO := -9, Raw_WRIO := 3269, H_Raw_RIO := 31208, L_Raw_WRIO := 3277, H_Raw_WRIO := 16383, HEU := 2, Hty := 1, AL := 1, ALL := 1, RIO_Hty := 1);
   LIT401_FB_01 : AIN_FBD;
   Logix_Status : Logix_Status_FP := (Set_FaceplateAnimation := 90, Val_ProductCode := 92, MemoryTemp[0] := 5, MemoryTemp[1] := 1, MemoryTemp[3] := 32290, MemoryTemp[4] := 3, MemoryTemp[5] := 18578, MemoryTemp[6] := 7, MemoryTemp[9] := 2, MemoryTemp[11] := -4608, MemoryTemp[12] := 3, MemoryTemp[14] := 8, MemoryTemp[17] := 5, MemoryTemp[21] := 6, MemoryTemp[23] := 32052, MemoryTemp[24] := 3, MemoryTemp[25] := 7, MemoryTemp[27] := 18376, MemoryTemp[28] := 7, Val_raw_data := 12384, Sts_IO_LED_raw := 2, Sts_ProductCode := 92, MemoryRequestData[0] := 5, MemoryRequestData[2] := 1, MemoryRequestData[4] := 2, MemoryRequestData[6] := 5, MemoryRequestData[8] := 6, MemoryRequestData[10] := 7, Sts_Run := 1, Sts_KS_in_remote := 1, Sts_Ladder_Working := 1, Set_Controller_Description := 'P6: RO Product System', UpdateDelayTimer.PRE := 1000, UpdateDelayTimer.ACC := 798, UpdateDelayTimer.EN := 1, UpdateDelayTimer.TT := 1, Val_MFS.timelow := 71751885, Val_MFS.timehigh := 206334, Val_MFS.type := 3, Val_MFS.code := 20, Val_MFS.info[1] := 1, Sts_IO_LED.FlashingGreen := 1, Sts_Battery_LED.Off := 1, MemoryData.Free_Mem_IO := 915592, MemoryData.Free_Mem_DT := 1909320, MemoryData.Total_Mem_IO := 1030144, MemoryData.Total_Mem_DT := 2097152, MemoryData.Biggest_IO_Mem_Size_Ava := 914640, MemoryData.Biggest_DT_Mem_Size_Ava := 1908512);
   LS401_FB : SWITCH_FBD;
   LSH601_FB : SWITCH_FBD := (Alarm := 1, Status := 1);
   LSH601_FB_01 : SWITCH_FBD;
   LSH601_FB_02 : SWITCH_FBD;
   LSH602_FB : SWITCH_FBD := (Alarm := 1, Status := 1);
   LSH603_FB : SWITCH_FBD;
   LSL601_FB : SWITCH_FBD;
   LSL601_FB_01 : SWITCH_FBD;
   LSL601_FB_02 : SWITCH_FBD;
   LSL601_FB_03 : SWITCH_FBD;
   LSL602_FB : SWITCH_FBD;
   LSL603_FB : SWITCH_FBD := (Alarm := 1, Status := 1);
   Memory_Message : MESSAGE;
        MessageParameters(ServiceCode := 16#0003, LocalElement := Logix_Status.MemoryRequestData[0], DestinationTag := Logix_Status.MemoryTemp[0], ...)
   MV301_FB : MV_FBD := (Cmd_Close := 1, Open_TM := 25, ZSC := 1, Close_TM := 25);
   MV302_FB : MV_FBD := (Cmd_Close := 1, Open_TM := 25, ZSC := 1, Close_TM := 25);
   MV303_FB : MV_FBD := (Cmd_Close := 1, Open_TM := 25, ZSC := 1, Close_TM := 25);
   MV304_FB : MV_FBD := (Cmd_Close := 1, Open_TM := 25, ZSC := 1, Close_TM := 25);
   P1_LIT101_MSG : MESSAGE;
        MessageParameters(ServiceCode := 16#004c, LocalElement := HMI_LIT101, ...)
   P201_FB : PMP_FBD;
   P202_FB : PMP_FBD;
   P2_AIT202_MSG : MESSAGE;
        MessageParameters(ServiceCode := 16#004c, LocalElement := HMI_AIT202, ...)
   P301_FB : PMP_FBD := (Remote := 1, Start_TM := 3, Stop_TM := 3, Permissive := -1);
   P302_FB : PMP_FBD := (Remote := 1, Start_TM := 3, Stop_TM := 3, Permissive := -1);
   P401_FB : PMP_FBD := (Remote := 1, Start_TM := 3, Stop_TM := 3, Permissive := -1);
   P401_FB_01 : PMP_FBD;
   P401_FB_02 : PMP_FBD;
   P402_FB : PMP_FBD := (Remote := 1, Start_TM := 3, Stop_TM := 3, Permissive := -1);
   P402_FB_01 : PMP_FBD;
   P403_FB : PMP_FBD := (Remote := 1, Start_TM := 3, Stop_TM := 3, Permissive := -1);
   P404_FB : PMP_FBD := (Remote := 1, Start_TM := 3, Stop_TM := 3, Permissive := -1);
   P601_FB : PMP_FBD := (Avl := 1, RunHr := 36.1, Total_RunHr := 36.1, Auto := 1, Remote := 1, Start_TM := 3, Stop_TM := 3, Rst := 1, Permissive := -1);
   P601_FB_01 : PMP_FBD;
   P601_FB_02 : PMP_FBD;
   P602_FB : PMP_FBD := (Avl := 1, RunHr := 1.05, Total_RunHr := 1.05, Auto := 1, Remote := 1, Start_TM := 3, Stop_TM := 3, Rst := 1, Permissive := -1);
   P603_FB : PMP_FBD := (Avl := 1, Auto := 1, Remote := 1, Start_TM := 3, Stop_TM := 3, Rst := 1, Permissive := -2, Shutdown := 1);
   P6_P602_AUTOINP : AUTOINP_UDT;
   P_NAHSO3_ORP_DUTY_FB : Duty2_FBD;
   P_RO_FEED_DUTY_FB : Duty2_FBD;
   P_RO_FEED_DUTY_FB_01 : Duty2_FBD;
   P_UF_FEED_DUTY_FB : Duty2_FBD := (AutoInp := 1);
   PLANT_CRITICAL_SD : AUTOINP_UDT;
   PSH301_FB : SWITCH_FBD;
   PSH301_FB_01 : SWITCH_FBD;
   REDUNDANT_STATUS : RED_STAT := (Redundancy_status_of_the_controller := 2, Redundancy_state_of_the_partner := 8);
   UV401_FB : UV_FBD := (AutoInp := 1, Remote := 1, Start_TM := 3, Stop_TM := 3, Permissive := -1);
   W_AI_AIT_401_HRDNSS : INT := 3266;
   W_AI_AIT_401_HRDNSS_HTY : BOOL;
   W_AI_AIT_402_ORP : INT := 3268;
   W_AI_AIT_402_ORP_HTY : BOOL;
   W_AI_DPIT_301_DPRESS : INT;
   W_AI_DPIT_301_DPRESS_HTY : BOOL;
   W_AI_FIT_301_FLOW : INT;
   W_AI_FIT_301_FLOW_HTY : BOOL;
   W_AI_FIT_401_FLOW : INT := 3263;
   W_AI_FIT_401_FLOW_HTY : BOOL;
   W_AI_FIT_601_FLOW : INT;
   W_AI_FIT_601_FLOW_HTY : BOOL := 1;
   W_AI_FIT_601_HTY : BOOL;
   W_AI_LIT_301_LEVEL : INT;
   W_AI_LIT_301_LEVEL_HTY : BOOL;
   W_AI_LIT_401_LEVEL : INT := 3269;
   W_AI_LIT_401_LEVEL_HTY : BOOL;
   W_AI_RIO6_SPARE_01 : INT;
   W_AI_RIO6_SPARE_01_HTY : BOOL := 1;
   XXX : DINT;
END_VAR

PROGRAM MainProgram   (* main routine MainRoutine *)
VAR
   FIT_FBD_01 : FIT_FBD;
   PMP_FBD_01 : PMP_FBD;
   SWITCH_FBD_01 : SWITCH_FBD;
END_VAR

ROUTINE IO   (* structured text *)
   (*DIGITAL INPUTS*)
   DI_WIFI_PLC_6	:=RIO6:0:I.Data.0;
   DI_WIFI_RIO_6	:=RIO6:0:I.Data.1;
   DI_P_601_AUTO	:=RIO6:0:I.Data.2;
   DI_P_601_RUN	:=RIO6:0:I.Data.3;
   DI_P_601_FAULT	:=RIO6:0:I.Data.4;
   DI_P_602_AUTO	:=RIO6:0:I.Data.5;
   DI_P_602_RUN	:=RIO6:0:I.Data.6;
   DI_P_602_FAULT	:=RIO6:0:I.Data.7;
   DI_P_603_AUTO	:=RIO6:0:I.Data.8;
   DI_P_603_RUN	:=RIO6:0:I.Data.9;
   DI_P_603_FAULT	:=RIO6:0:I.Data.10;
   DI_LS_601_LOW	:=RIO6:0:I.Data.11;
   DI_LS_601_HIGH	:=RIO6:0:I.Data.12;
   DI_LS_602_LOW	:=RIO6:0:I.Data.13;
   DI_LS_602_HIGH	:=RIO6:0:I.Data.14;
   DI_LS_603_LOW	:=RIO6:0:I.Data.15;
   DI_LS_603_HIGH	:=RIO6:0:I.Data.16;
   DI_RIO6_SPARE_17:=RIO6:0:I.Data.17;
   DI_RIO6_SPARE_18:=RIO6:0:I.Data.18;
   DI_RIO6_SPARE_19:=RIO6:0:I.Data.19;
   DI_RIO6_SPARE_20:=RIO6:0:I.Data.20;
   DI_RIO6_SPARE_21:=RIO6:0:I.Data.21;
   DI_RIO6_SPARE_22:=RIO6:0:I.Data.22;
   DI_RIO6_SPARE_23:=RIO6:0:I.Data.23;
   DI_RIO6_SPARE_24:=RIO6:0:I.Data.24;
   DI_RIO6_SPARE_25:=RIO6:0:I.Data.25;
   DI_RIO6_SPARE_26:=RIO6:0:I.Data.26;
   DI_RIO6_SPARE_27:=RIO6:0:I.Data.27;
   DI_RIO6_SPARE_28:=RIO6:0:I.Data.28;
   DI_RIO6_SPARE_29:=RIO6:0:I.Data.29;
   DI_RIO6_SPARE_30:=RIO6:0:I.Data.30;
   DI_RIO6_SPARE_31:=RIO6:0:I.Data.31;
   
   (*DIGITAL OUTPUTS*)
   RIO6:1:O.0	:=DO_P_601_START;
   RIO6:1:O.1	:=DO_P_602_START;
   RIO6:1:O.2	:=DO_P_603_START;
   RIO6:1:O.4	:=DO_RIO6_SPARE_04;
   RIO6:1:O.5	:=DO_RIO6_SPARE_05;
   RIO6:1:O.6	:=DO_RIO6_SPARE_06;
   RIO6:1:O.7	:=DO_RIO6_SPARE_07;
   RIO6:1:O.8	:=DO_RIO6_SPARE_08;
   RIO6:1:O.9	:=DO_RIO6_SPARE_09;
   RIO6:1:O.10	:=DO_RIO6_SPARE_10;
   RIO6:1:O.11	:=DO_RIO6_SPARE_11;
   RIO6:1:O.12	:=DO_RIO6_SPARE_12;
   RIO6:1:O.13	:=DO_RIO6_SPARE_13;
   RIO6:1:O.14	:=DO_RIO6_SPARE_14;
   RIO6:1:O.15	:=DO_RIO6_SPARE_15;
   
   (*ANALOG INPUTS*)
   AI_FIT_601_FLOW		:=RIO6:2:I.Ch0Data;
   AI_RIO6_SPARE_01	:=RIO6:2:I.Ch1Data;
   AI_RIO6_SPARE_02	:=RIO6:2:I.Ch2Data;
   AI_RIO6_SPARE_03	:=RIO6:2:I.Ch3Data;
   AI_RIO6_SPARE_04	:=RIO6:2:I.Ch4Data;
   AI_RIO6_SPARE_05	:=RIO6:2:I.Ch5Data;
   AI_RIO6_SPARE_06	:=RIO6:2:I.Ch6Data;
   AI_RIO6_SPARE_07	:=RIO6:2:I.Ch7Data;
   AI_RIO6_SPARE_08	:=RIO6:2:I.Ch8Data;
   AI_RIO6_SPARE_09	:=RIO6:2:I.Ch9Data;
   AI_RIO6_SPARE_10	:=RIO6:2:I.Ch10Data;
   AI_RIO6_SPARE_11	:=RIO6:2:I.Ch11Data;
   
   AI_FIT_601_FLOW_HTY		:=(NOT RIO6:2:I.GeneralFault);
   AI_RIO6_SPARE_01_HTY	:=(NOT RIO6:2:I.GeneralFault);
   AI_RIO6_SPARE_02_HTY	:=(NOT RIO6:2:I.GeneralFault);
   AI_RIO6_SPARE_03_HTY	:=(NOT RIO6:2:I.GeneralFault);
   AI_RIO6_SPARE_04_HTY	:=(NOT RIO6:2:I.GeneralFault);
   AI_RIO6_SPARE_05_HTY	:=(NOT RIO6:2:I.GeneralFault);
   AI_RIO6_SPARE_06_HTY	:=(NOT RIO6:2:I.GeneralFault);
   AI_RIO6_SPARE_07_HTY	:=(NOT RIO6:2:I.GeneralFault);
   AI_RIO6_SPARE_08_HTY	:=(NOT RIO6:2:I.GeneralFault);
   AI_RIO6_SPARE_09_HTY	:=(NOT RIO6:2:I.GeneralFault);
   AI_RIO6_SPARE_10_HTY	:=(NOT RIO6:2:I.GeneralFault);
   AI_RIO6_SPARE_11_HTY	:=(NOT RIO6:2:I.GeneralFault);
   
   (*WIRELESS ANALOG INPUTS*)
   W_AI_FIT_601_FLOW		:=WRIO6:1:I.Ch0Data;
   W_AI_RIO6_SPARE_01		:=WRIO6:1:I.Ch1Data;
   
   W_AI_FIT_601_FLOW_HTY	:=(NOT WRIO6:1:I.Ch0Fault);
   W_AI_RIO6_SPARE_01_HTY	:=(NOT WRIO6:1:I.Ch1Fault);
   
   (*Wireless Selction*)
   HMI_WIFI.PLC_WIFI		:= DI_WIFI_PLC_6;
   HMI_WIFI.RIO_WIFI		:= DI_WIFI_RIO_6;
END_ROUTINE

ROUTINE Logix_Status   (* ladder *)
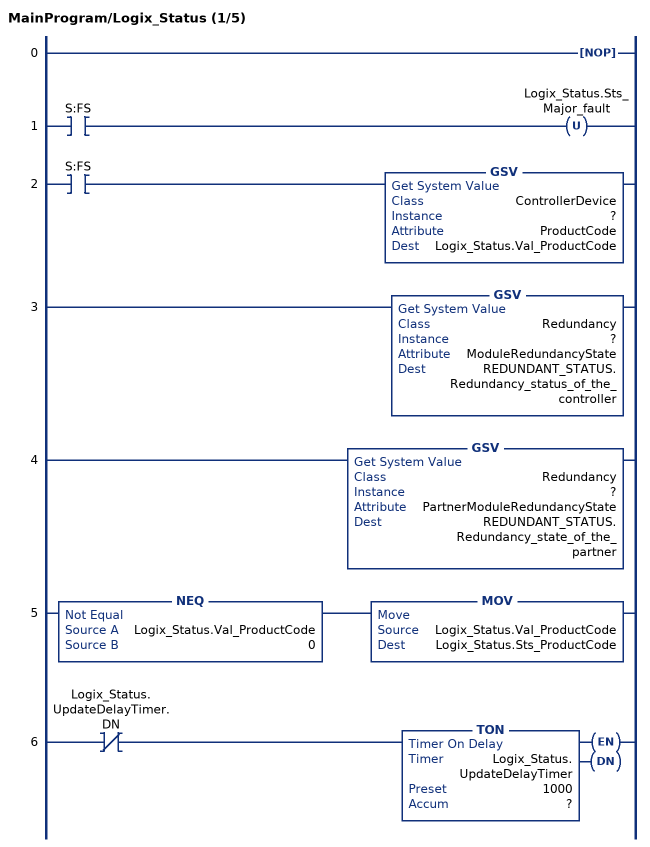
   0: NOP();
   1: XIC(S:FS)OTU(Logix_Status.Sts_Major_fault);
   2: XIC(S:FS)GSV(ControllerDevice,?,ProductCode,Logix_Status.Val_ProductCode);
   3: GSV(Redundancy,?,ModuleRedundancyState,REDUNDANT_STATUS.Redundancy_status_of_the_controller);
   4: GSV(Redundancy,?,PartnerModuleRedundancyState,REDUNDANT_STATUS.Redundancy_state_of_the_partner);
   5: NEQ(Logix_Status.Val_ProductCode,0)MOV(Logix_Status.Val_ProductCode,Logix_Status.Sts_ProductCode);
   6: XIO(Logix_Status.UpdateDelayTimer.DN)TON(Logix_Status.UpdateDelayTimer,?,?);
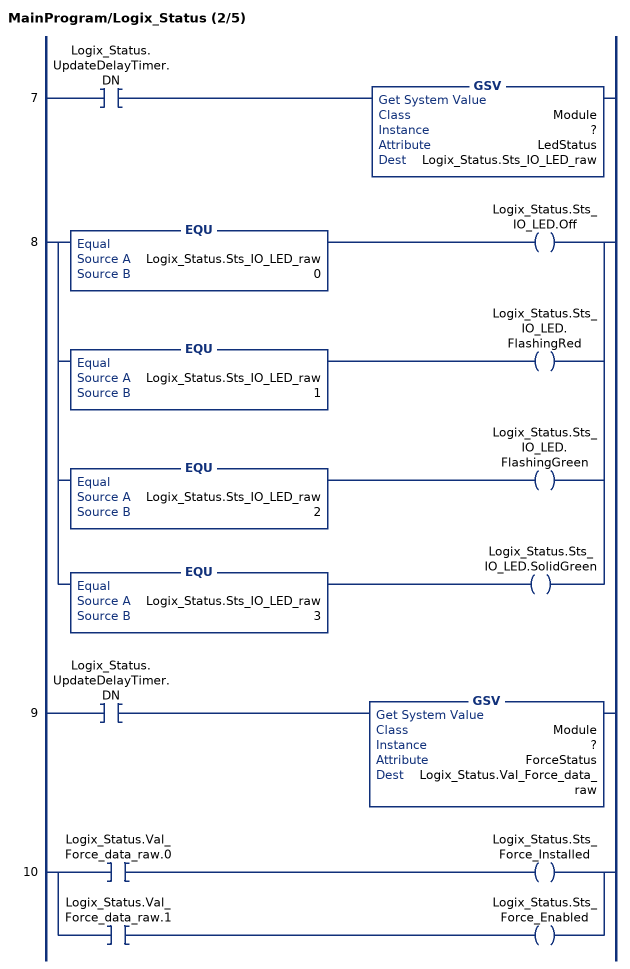
   7: XIC(Logix_Status.UpdateDelayTimer.DN)GSV(Module,?,LedStatus,Logix_Status.Sts_IO_LED_raw);
   8: [EQU(Logix_Status.Sts_IO_LED_raw,0) OTE(Logix_Status.Sts_IO_LED.Off) ,EQU(Logix_Status.Sts_IO_LED_raw,1) OTE(Logix_Status.Sts_IO_LED.FlashingRed) ,EQU(Logix_Status.Sts_IO_LED_raw,2) OTE(Logix_Status.Sts_IO_LED.FlashingGreen) ,EQU(Logix_Status.Sts_IO_LED_raw,3) OTE(Logix_Status.Sts_IO_LED.SolidGreen) ];
   9: XIC(Logix_Status.UpdateDelayTimer.DN)GSV(Module,?,ForceStatus,Logix_Status.Val_Force_data_raw);
   10: [XIC(Logix_Status.Val_Force_data_raw.0) OTE(Logix_Status.Sts_Force_Installed) ,XIC(Logix_Status.Val_Force_data_raw.1) OTE(Logix_Status.Sts_Force_Enabled) ];
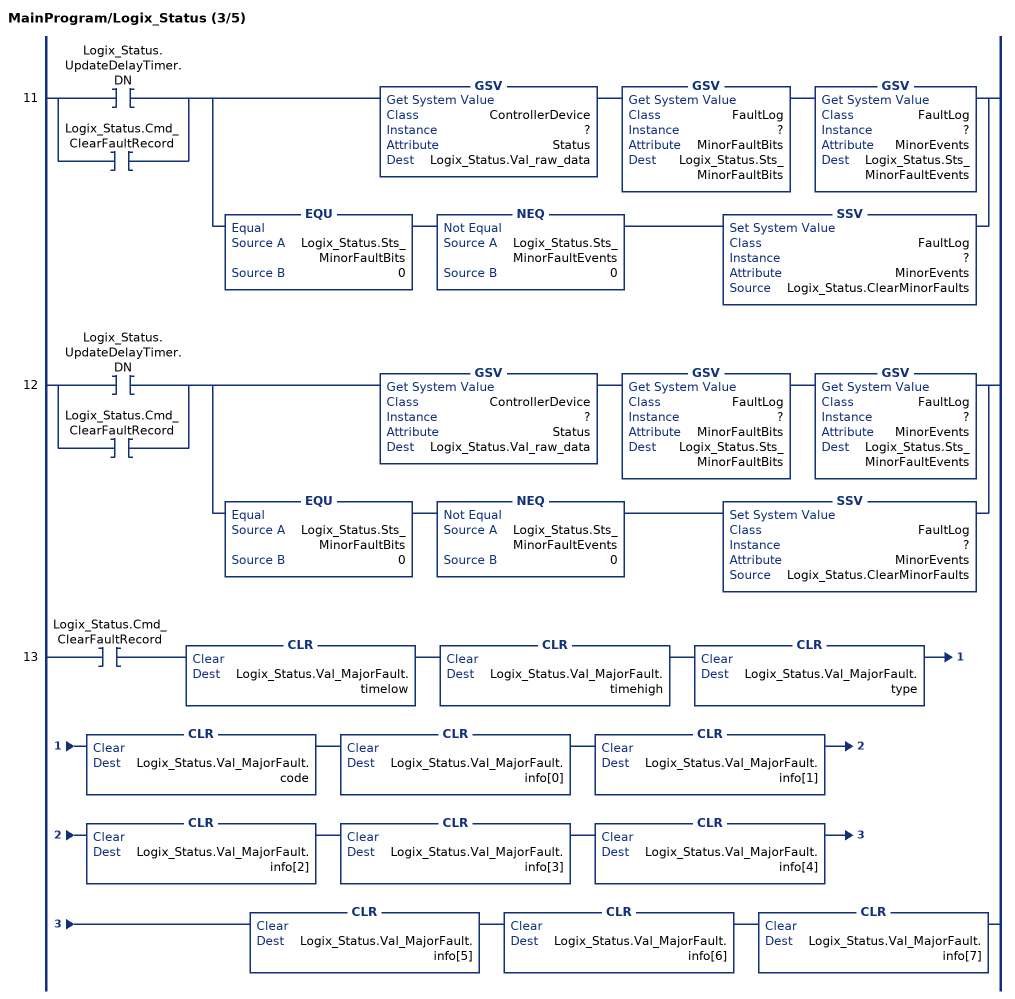
   11: [XIC(Logix_Status.UpdateDelayTimer.DN) ,XIC(Logix_Status.Cmd_ClearFaultRecord) ][GSV(ControllerDevice,?,Status,Logix_Status.Val_raw_data) GSV(FaultLog,?,MinorFaultBits,Logix_Status.Sts_MinorFaultBits) GSV(FaultLog,?,MinorEvents,Logix_Status.Sts_MinorFaultEvents) ,EQU(Logix_Status.Sts_MinorFaultBits,0) NEQ(Logix_Status.Sts_MinorFaultEvents,0) SSV(FaultLog,?,MinorEvents,Logix_Status.ClearMinorFaults) ];
   12: [XIC(Logix_Status.UpdateDelayTimer.DN) ,XIC(Logix_Status.Cmd_ClearFaultRecord) ][GSV(ControllerDevice,?,Status,Logix_Status.Val_raw_data) GSV(FaultLog,?,MinorFaultBits,Logix_Status.Sts_MinorFaultBits) GSV(FaultLog,?,MinorEvents,Logix_Status.Sts_MinorFaultEvents) ,EQU(Logix_Status.Sts_MinorFaultBits,0) NEQ(Logix_Status.Sts_MinorFaultEvents,0) SSV(FaultLog,?,MinorEvents,Logix_Status.ClearMinorFaults) ];
   13: XIC(Logix_Status.Cmd_ClearFaultRecord)CLR(Logix_Status.Val_MajorFault.timelow)CLR(Logix_Status.Val_MajorFault.timehigh)CLR(Logix_Status.Val_MajorFault.type)CLR(Logix_Status.Val_MajorFault.code)CLR(Logix_Status.Val_MajorFault.info[0])CLR(Logix_Status.Val_MajorFault.info[1])CLR(Logix_Status.Val_MajorFault.info[2])CLR(Logix_Status.Val_MajorFault.info[3])CLR(Logix_Status.Val_MajorFault.info[4])CLR(Logix_Status.Val_MajorFault.info[5])CLR(Logix_Status.Val_MajorFault.info[6])CLR(Logix_Status.Val_MajorFault.info[7]);
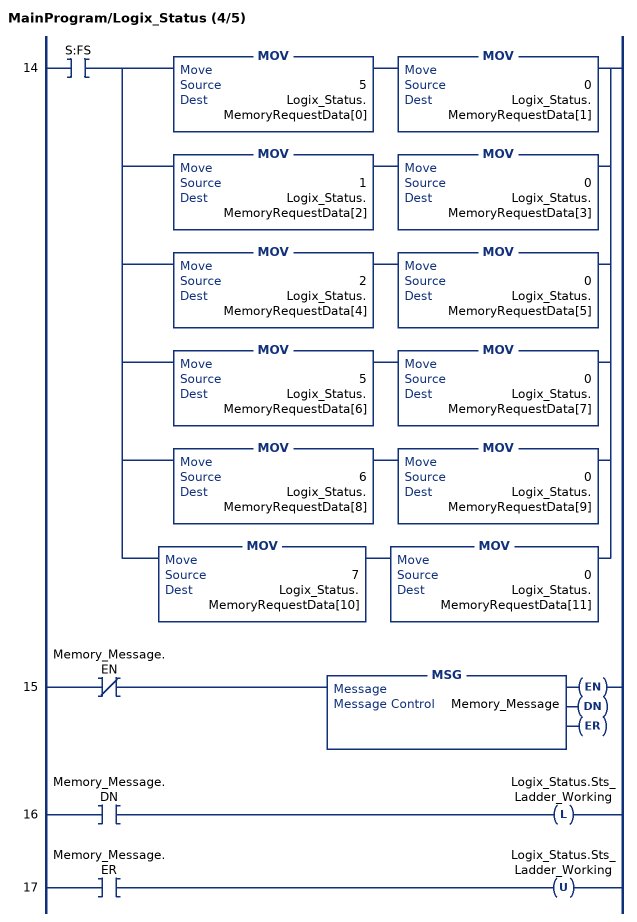
   14: XIC(S:FS)[MOV(5,Logix_Status.MemoryRequestData[0]) MOV(0,Logix_Status.MemoryRequestData[1]) ,MOV(1,Logix_Status.MemoryRequestData[2]) MOV(0,Logix_Status.MemoryRequestData[3]) ,MOV(2,Logix_Status.MemoryRequestData[4]) MOV(0,Logix_Status.MemoryRequestData[5]) ,MOV(5,Logix_Status.MemoryRequestData[6]) MOV(0,Logix_Status.MemoryRequestData[7]) ,MOV(6,Logix_Status.MemoryRequestData[8]) MOV(0,Logix_Status.MemoryRequestData[9]) ,MOV(7,Logix_Status.MemoryRequestData[10]) MOV(0,Logix_Status.MemoryRequestData[11]) ];
   15: XIO(Memory_Message.EN)MSG(Memory_Message);
   16: XIC(Memory_Message.DN)OTL(Logix_Status.Sts_Ladder_Working);
   17: XIC(Memory_Message.ER)OTU(Logix_Status.Sts_Ladder_Working);
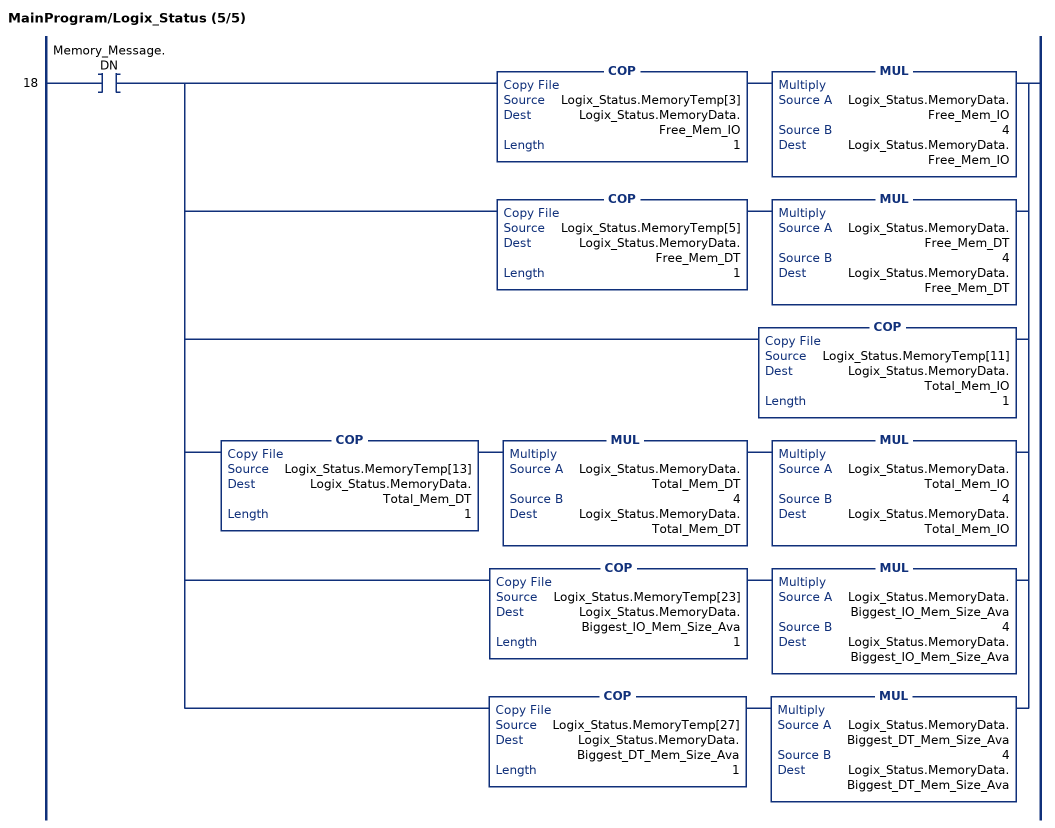
   18: XIC(Memory_Message.DN)[COP(Logix_Status.MemoryTemp[3],Logix_Status.MemoryData.Free_Mem_IO,1) MUL(Logix_Status.MemoryData.Free_Mem_IO,4,Logix_Status.MemoryData.Free_Mem_IO) ,COP(Logix_Status.MemoryTemp[5],Logix_Status.MemoryData.Free_Mem_DT,1) MUL(Logix_Status.MemoryData.Free_Mem_DT,4,Logix_Status.MemoryData.Free_Mem_DT) ,COP(Logix_Status.MemoryTemp[11],Logix_Status.MemoryData.Total_Mem_IO,1) ,COP(Logix_Status.MemoryTemp[13],Logix_Status.MemoryData.Total_Mem_DT,1) MUL(Logix_Status.MemoryData.Total_Mem_DT,4,Logix_Status.MemoryData.Total_Mem_DT) MUL(Logix_Status.MemoryData.Total_Mem_IO,4,Logix_Status.MemoryData.Total_Mem_IO) ,COP(Logix_Status.MemoryTemp[23],Logix_Status.MemoryData.Biggest_IO_Mem_Size_Ava,1) MUL(Logix_Status.MemoryData.Biggest_IO_Mem_Size_Ava,4,Logix_Status.MemoryData.Biggest_IO_Mem_Size_Ava) ,COP(Logix_Status.MemoryTemp[27],Logix_Status.MemoryData.Biggest_DT_Mem_Size_Ava,1) MUL(Logix_Status.MemoryData.Biggest_DT_Mem_Size_Ava,4,Logix_Status.MemoryData.Biggest_DT_Mem_Size_Ava) ];
END_ROUTINE

ROUTINE Main_Seq   (* structured text *)
   (*
   IF HMI_PLANT.STOP THEN
   	HMI_P6_STATE:=1;
   END_IF;
   *)
   
   IF HMI_PLANT.STOP OR PLANT_CRITICAL_SD.ON THEN
   	HMI_P6_STATE:=1;
   END_IF;
   
   
   
   
   
   
   _P602_AutoInp := P6_P602_AUTOINP.ON;
   
   (*
   if S:FS then
   	HMI_P6_STATE := 1;
   end_if;
   *)
   
   
   (*-----------WRITE FAULT CONDITION--------------*)
   
   CASE HMI_P6_STATE OF
   	1:(*PLANT IN STANDBY*)
   		_P601_AutoInp	:= 0;  (*RO PERMEATE*)
   		_P602_AutoInp	:= 0;  (*UF BACKWASH*)
   		_P603_AutoInp	:= 0;  (*CIP*)
   
   		IF HMI_P6_PERMISSIVE.ON AND HMI_PLANT.START THEN
   			HMI_P6_STATE:=2;
   		END_IF;
   
   	2:(*PLANT IN STANDBY*)
   		_P_PERMEATE_SR.EnableIn				:= 1;
   		_P_PERMEATE_SR.Set					:= HMI_LSH601.Alarm AND HMI_AIT202.Pv >= 7 AND NOT HMI_LIT101.AHH AND 0  ;
   	(*	_P_PERMEATE_SR.Set					:= HMI_LSH601.Alarm AND HMI_AIT202.Pv >= 7 AND NOT HMI_LIT101.AHH;*)
   		_P_PERMEATE_SR.Reset				:= HMI_LIT101.AHH OR HMI_LSL601.Alarm OR HMI_AIT202.Pv < 7 ;
   		SETD( _P_PERMEATE_SR);
   		_P601_AutoInp						:= _P_PERMEATE_SR.Out;
   
   		_P602_AutoInp	:= _P602_AutoInp; (*SIGNAL FROM P3, UF*)
   		_P603_AutoInp	:= _P603_AutoInp; (*SIGNAL FROM P5, RO*)
   
   ELSE
   	HMI_P6_STATE:=1;
   END_CASE;
END_ROUTINE

ROUTINE MainRoutine   (* ladder *)
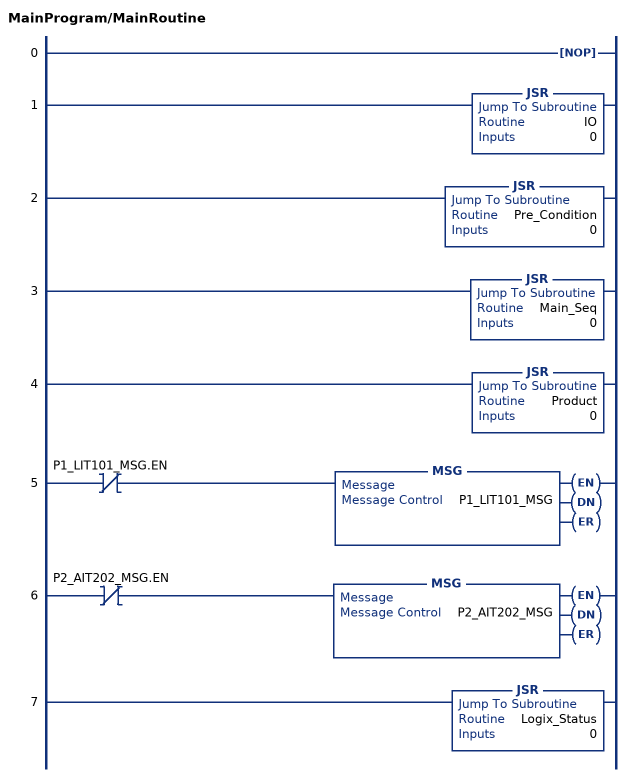
   0: NOP();
   1: JSR(IO,0);
   2: JSR(Pre_Condition,0);
   3: JSR(Main_Seq,0);
   4: JSR(Product,0);
   5: XIO(P1_LIT101_MSG.EN)MSG(P1_LIT101_MSG);
   6: XIO(P2_AIT202_MSG.EN)MSG(P2_AIT202_MSG);
   7: JSR(Logix_Status,0);
END_ROUTINE

ROUTINE Pre_Condition   (* structured text *)
   IF HMI_PLANT_RESET.ON THEN
   	HMI_P601.Reset	:=1;
   	HMI_P602.Reset	:=1;
   	HMI_P603.Reset	:=1;
   END_IF;
   
   (*ALL INSTRUMENT IN AUTO MODE*)
   IF HMI_PLANT_AUTO.ON THEN
   	HMI_P601.Auto	:=1;
   	HMI_P602.Auto	:=1;
   	HMI_P603.Auto	:=1;
   END_IF;
   
   (*ALL INSTRUMENT IN MANUAL MODE*)
   IF HMI_PLANT_AUTO.OFF THEN
   	HMI_P601.Auto	:=0;
   	HMI_P602.Auto	:=0;
   	HMI_P603.Auto	:=0;
   END_IF;
   
   HMI_P6_PERMISSIVE.ON:= HMI_P601.Avl AND HMI_P602.Avl (*AND HMI_P603.Avl*);
   
   _FIT601_Tot_Enb	:= HMI_P602.status=2;
   
   (*P601 Permissive*)
   HMI_P601.Permissive.0 	:= NOT HMI_LSL601.Alarm;
   HMI_P601.Permissive.1 	:= 1;
   HMI_P601.Permissive.2 	:= 1;
   HMI_P601.Permissive.3 	:= 1;
   HMI_P601.Permissive.4 	:= 1;
   HMI_P601.Permissive.5 	:= 1;
   HMI_P601.Permissive.6 	:= 1;
   HMI_P601.Permissive.7 	:= 1;
   HMI_P601.Permissive.8 	:= 1;
   HMI_P601.Permissive.9 	:= 1;
   HMI_P601.Permissive.10 	:= 1;
   HMI_P601.Permissive.11 	:= 1;
   HMI_P601.Permissive.12 	:= 1;
   HMI_P601.Permissive.13	:= 1;
   HMI_P601.Permissive.14	:= 1;
   HMI_P601.Permissive.15 	:= 1;
   
   HMI_P601_MSG.PERMISSIVE1 := HMI_P601.Permissive.0;
   HMI_P601_MSG.PERMISSIVE2 := 0;
   HMI_P601_MSG.PERMISSIVE3 := 0;
   HMI_P601_MSG.PERMISSIVE4 := 0;
   HMI_P601_MSG.PERMISSIVE5 := 0;
   
   (*P602 Permissive*)
   HMI_P602.Permissive.0 	:= NOT HMI_LSL602.Alarm;
   HMI_P602.Permissive.1 	:= 1;
   HMI_P602.Permissive.2 	:= 1;
   HMI_P602.Permissive.3 	:= 1;
   HMI_P602.Permissive.4 	:= 1;
   HMI_P602.Permissive.5 	:= 1;
   HMI_P602.Permissive.6 	:= 1;
   HMI_P602.Permissive.7 	:= 1;
   HMI_P602.Permissive.8 	:= 1;
   HMI_P602.Permissive.9 	:= 1;
   HMI_P602.Permissive.10 	:= 1;
   HMI_P602.Permissive.11 	:= 1;
   HMI_P602.Permissive.12 	:= 1;
   HMI_P602.Permissive.13	:= 1;
   HMI_P602.Permissive.14	:= 1;
   HMI_P602.Permissive.15 	:= 1;
   
   HMI_P602_MSG.PERMISSIVE1 := HMI_P602.Permissive.0;
   HMI_P602_MSG.PERMISSIVE2 := 0;
   HMI_P602_MSG.PERMISSIVE3 := 0;
   HMI_P602_MSG.PERMISSIVE4 := 0;
   HMI_P602_MSG.PERMISSIVE5 := 0;
   
   (*P603 Permissive*)
   HMI_P603.Permissive.0 	:= NOT HMI_LSL603.Alarm;
   HMI_P603.Permissive.1 	:= 1;
   HMI_P603.Permissive.2 	:= 1;
   HMI_P603.Permissive.3 	:= 1;
   HMI_P603.Permissive.4 	:= 1;
   HMI_P603.Permissive.5 	:= 1;
   HMI_P603.Permissive.6 	:= 1;
   HMI_P603.Permissive.7 	:= 1;
   HMI_P603.Permissive.8 	:= 1;
   HMI_P603.Permissive.9 	:= 1;
   HMI_P603.Permissive.10 	:= 1;
   HMI_P603.Permissive.11 	:= 1;
   HMI_P603.Permissive.12 	:= 1;
   HMI_P603.Permissive.13	:= 1;
   HMI_P603.Permissive.14	:= 1;
   HMI_P603.Permissive.15 	:= 1;
   
   HMI_P603_MSG.PERMISSIVE1 := HMI_P603.Permissive.0;
   HMI_P603_MSG.PERMISSIVE2 := 0;
   HMI_P603_MSG.PERMISSIVE3 := 0;
   HMI_P603_MSG.PERMISSIVE4 := 0;
   HMI_P603_MSG.PERMISSIVE5 := 0;
   
   (*-------------------------------------------------------------------------------------*)
   (*P601 Shutdown*)
   HMI_P601.SD.0 	:= HMI_LSL601.Alarm;
   HMI_P601.SD.1 	:= 0;
   HMI_P601.SD.2 	:= 0;
   HMI_P601.SD.3 	:= 0;
   HMI_P601.SD.4 	:= 0;
   HMI_P601.SD.5 	:= 0;
   HMI_P601.SD.6 	:= 0;
   HMI_P601.SD.7 	:= 0;
   HMI_P601.SD.8 	:= 0;
   HMI_P601.SD.9 	:= 0;
   HMI_P601.SD.10 	:= 0;
   HMI_P601.SD.11 	:= 0;
   HMI_P601.SD.12 	:= 0;
   HMI_P601.SD.13 	:= 0;
   HMI_P601.SD.14 	:= 0;
   HMI_P601.SD.15 	:= 0;
   
   HMI_P601_MSG.SHUTDOWN1 := HMI_P601.SHUTDOWN.0 ;
   HMI_P601_MSG.SHUTDOWN2 := HMI_P601.SHUTDOWN.1 ;
   HMI_P601_MSG.SHUTDOWN3 := HMI_P601.SHUTDOWN.2 ;
   HMI_P601_MSG.SHUTDOWN4 := HMI_P601.SHUTDOWN.3 ;
   HMI_P601_MSG.SHUTDOWN5 := HMI_P601.SHUTDOWN.4 ;
   
   (*P602 Shutdown*)
   HMI_P602.SD.0 	:= 0;(*HMI_LSL602.Alarm;*)
   HMI_P602.SD.1 	:= 0;
   HMI_P602.SD.2 	:= 0;
   HMI_P602.SD.3 	:= 0;
   HMI_P602.SD.4 	:= 0;
   HMI_P602.SD.5 	:= 0;
   HMI_P602.SD.6 	:= 0;
   HMI_P602.SD.7 	:= 0;
   HMI_P602.SD.8 	:= 0;
   HMI_P602.SD.9 	:= 0;
   HMI_P602.SD.10 	:= 0;
   HMI_P602.SD.11 	:= 0;
   HMI_P602.SD.12 	:= 0;
   HMI_P602.SD.13 	:= 0;
   HMI_P602.SD.14 	:= 0;
   HMI_P602.SD.15 	:= 0;
   
   HMI_P602_MSG.SHUTDOWN1 := HMI_P602.SHUTDOWN.0 ;
   HMI_P602_MSG.SHUTDOWN2 := HMI_P602.SHUTDOWN.1 ;
   HMI_P602_MSG.SHUTDOWN3 := HMI_P602.SHUTDOWN.2 ;
   HMI_P602_MSG.SHUTDOWN4 := HMI_P602.SHUTDOWN.3 ;
   HMI_P602_MSG.SHUTDOWN5 := HMI_P602.SHUTDOWN.4 ;
   
   (*P603 Shutdown*)
   HMI_P603.SD.0 	:= HMI_LSL603.Alarm;
   HMI_P603.SD.1 	:= 0;
   HMI_P603.SD.2 	:= 0;
   HMI_P603.SD.3 	:= 0;
   HMI_P603.SD.4 	:= 0;
   HMI_P603.SD.5 	:= 0;
   HMI_P603.SD.6 	:= 0;
   HMI_P603.SD.7 	:= 0;
   HMI_P603.SD.8 	:= 0;
   HMI_P603.SD.9 	:= 0;
   HMI_P603.SD.10 	:= 0;
   HMI_P603.SD.11 	:= 0;
   HMI_P603.SD.12 	:= 0;
   HMI_P603.SD.13 	:= 0;
   HMI_P603.SD.14 	:= 0;
   HMI_P603.SD.15 	:= 0;
   
   HMI_P603_MSG.SHUTDOWN1 := HMI_P603.SHUTDOWN.0 ;
   HMI_P603_MSG.SHUTDOWN2 := HMI_P603.SHUTDOWN.1 ;
   HMI_P603_MSG.SHUTDOWN3 := HMI_P603.SHUTDOWN.2 ;
   HMI_P603_MSG.SHUTDOWN4 := HMI_P603.SHUTDOWN.3 ;
   HMI_P603_MSG.SHUTDOWN5 := HMI_P603.SHUTDOWN.4 ;
END_ROUTINE

ROUTINE Product   (* function block diagram *)
   SHEET 1
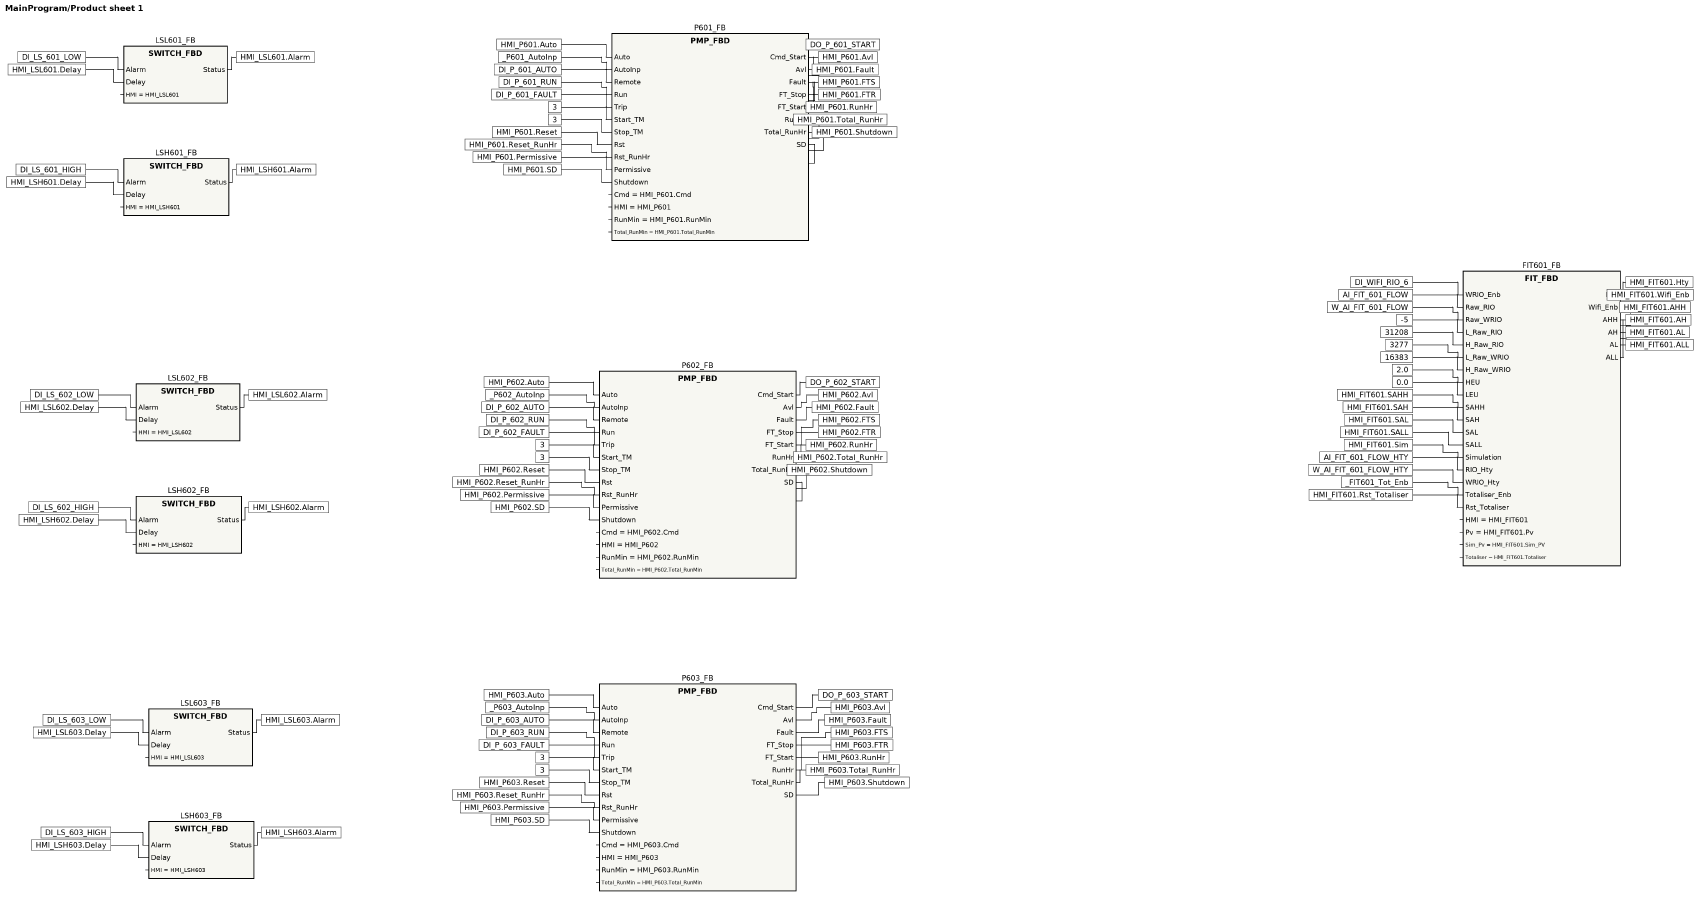
   LSL601_FB : SWITCH_FBD(Alarm := DI_LS_601_LOW, Delay := HMI_LSL601.Delay, HMI := HMI_LSL601);
   LSH601_FB : SWITCH_FBD(Alarm := DI_LS_601_HIGH, Delay := HMI_LSH601.Delay, HMI := HMI_LSH601);
   LSL602_FB : SWITCH_FBD(Alarm := DI_LS_602_LOW, Delay := HMI_LSL602.Delay, HMI := HMI_LSL602);
   LSH602_FB : SWITCH_FBD(Alarm := DI_LS_602_HIGH, Delay := HMI_LSH602.Delay, HMI := HMI_LSH602);
   LSL603_FB : SWITCH_FBD(Alarm := DI_LS_603_LOW, Delay := HMI_LSL603.Delay, HMI := HMI_LSL603);
   LSH603_FB : SWITCH_FBD(Alarm := DI_LS_603_HIGH, Delay := HMI_LSH603.Delay, HMI := HMI_LSH603);
   HMI_LSL601.Alarm := LSL601_FB.Status;
   HMI_LSH601.Alarm := LSH601_FB.Status;
   HMI_LSL602.Alarm := LSL602_FB.Status;
   HMI_LSH602.Alarm := LSH602_FB.Status;
   HMI_LSL603.Alarm := LSL603_FB.Status;
   HMI_LSH603.Alarm := LSH603_FB.Status;
   P602_FB : PMP_FBD(Auto := HMI_P602.Auto, AutoInp := _P602_AutoInp, Remote := DI_P_602_AUTO, Run := DI_P_602_RUN, Trip := DI_P_602_FAULT, Start_TM := 3, Stop_TM := 3, Rst := HMI_P602.Reset, Rst_RunHr := HMI_P602.Reset_RunHr, Permissive := HMI_P602.Permissive, Shutdown := HMI_P602.SD, Cmd := HMI_P602.Cmd, HMI := HMI_P602, RunMin := HMI_P602.RunMin, Total_RunMin := HMI_P602.Total_RunMin);
   P603_FB : PMP_FBD(Auto := HMI_P603.Auto, AutoInp := _P603_AutoInp, Remote := DI_P_603_AUTO, Run := DI_P_603_RUN, Trip := DI_P_603_FAULT, Start_TM := 3, Stop_TM := 3, Rst := HMI_P603.Reset, Rst_RunHr := HMI_P603.Reset_RunHr, Permissive := HMI_P603.Permissive, Shutdown := HMI_P603.SD, Cmd := HMI_P603.Cmd, HMI := HMI_P603, RunMin := HMI_P603.RunMin, Total_RunMin := HMI_P603.Total_RunMin);
   P601_FB : PMP_FBD(Auto := HMI_P601.Auto, AutoInp := _P601_AutoInp, Remote := DI_P_601_AUTO, Run := DI_P_601_RUN, Trip := DI_P_601_FAULT, Start_TM := 3, Stop_TM := 3, Rst := HMI_P601.Reset, Rst_RunHr := HMI_P601.Reset_RunHr, Permissive := HMI_P601.Permissive, Shutdown := HMI_P601.SD, Cmd := HMI_P601.Cmd, HMI := HMI_P601, RunMin := HMI_P601.RunMin, Total_RunMin := HMI_P601.Total_RunMin);
   HMI_P602.Shutdown := P602_FB.SD;
   HMI_P601.Total_RunHr := P601_FB.Total_RunHr;
   HMI_P602.Total_RunHr := P602_FB.Total_RunHr;
   DO_P_601_START := P601_FB.Cmd_Start;
   HMI_P601.RunHr := P601_FB.RunHr;
   DO_P_602_START := P602_FB.Cmd_Start;
   HMI_P602.RunHr := P602_FB.RunHr;
   HMI_P603.Total_RunHr := P603_FB.Total_RunHr;
   HMI_P601.Fault := P601_FB.Fault;
   HMI_P601.Shutdown := P601_FB.SD;
   HMI_P602.Fault := P602_FB.Fault;
   HMI_P601.Avl := P601_FB.Avl;
   HMI_P601.FTS := P601_FB.FT_Stop;
   HMI_P601.FTR := P601_FB.FT_Start;
   HMI_P602.Avl := P602_FB.Avl;
   HMI_P602.FTS := P602_FB.FT_Stop;
   HMI_P602.FTR := P602_FB.FT_Start;
   DO_P_603_START := P603_FB.Cmd_Start;
   HMI_P603.RunHr := P603_FB.RunHr;
   HMI_P603.Fault := P603_FB.Fault;
   HMI_P603.Shutdown := P603_FB.SD;
   HMI_P603.Avl := P603_FB.Avl;
   HMI_P603.FTS := P603_FB.FT_Stop;
   HMI_P603.FTR := P603_FB.FT_Start;
   FIT601_FB : FIT_FBD(WRIO_Enb := DI_WIFI_RIO_6, Raw_RIO := AI_FIT_601_FLOW, Raw_WRIO := W_AI_FIT_601_FLOW, L_Raw_RIO := -5, H_Raw_RIO := 31208, L_Raw_WRIO := 3277, H_Raw_WRIO := 16383, HEU := 2.0, LEU := 0.0, SAHH := HMI_FIT601.SAHH, SAH := HMI_FIT601.SAH, SAL := HMI_FIT601.SAL, SALL := HMI_FIT601.SALL, Simulation := HMI_FIT601.Sim, RIO_Hty := AI_FIT_601_FLOW_HTY, WRIO_Hty := W_AI_FIT_601_FLOW_HTY, Totaliser_Enb := _FIT601_Tot_Enb, Rst_Totaliser := HMI_FIT601.Rst_Totaliser, HMI := HMI_FIT601, Pv := HMI_FIT601.Pv, Sim_Pv := HMI_FIT601.Sim_PV, Totaliser := HMI_FIT601.Totaliser);
   HMI_FIT601.Wifi_Enb := FIT601_FB.Wifi_Enb;
   HMI_FIT601.AHH := FIT601_FB.AHH;
   HMI_FIT601.Hty := FIT601_FB.Hty;
   HMI_FIT601.AH := FIT601_FB.AH;
   HMI_FIT601.AL := FIT601_FB.AL;
   HMI_FIT601.ALL := FIT601_FB.ALL;
END_ROUTINE
END_PROGRAM
